(* Logix 5000 project; controller reports 1756-L63 rev 20.11; software revision 20.04; part 3 of 52 *)

        [200].log_data[5].valid := 1, [200].log_data[6].valid := 1, [200].log_data[7].valid := 1, [200].log_data[8].valid := 1, [200].log_data[9].valid := 1, [200].log_data[10].valid := 1, [200].log_data[11].valid := 1, [200].log_data[12].valid := 1, [200].log_data[13].valid := 1, [200].log_data[14].valid := 1, [200].log_data[15].valid := 1, [200].log_data[16].valid := 1, [200].log_data[17].valid := 1, [200].log_data[18].valid := 1, [200].log_data[19].valid := 1, [200].time.Year := 2023, [200].time.Month := 1, [200].time.Day := 18, [200].time.Hour := 2, [200].time.Minute := 29, [200].time.Second := 59, [201].log_data[0].min := 1.0, [201].log_data[0].max := 1.0, [201].log_data[0].total := 900.0, [201].log_data[0].time := 900.0, [201].log_data[0].minminute := 30, [201].log_data[0].maxminute := 30, [201].log_data[0].valid := 1, [201].log_data[1].valid := 1, [201].log_data[2].valid := 1, [201].log_data[3].valid := 1, [201].log_data[4].valid := 1, [201].log_data[5].valid := 1, [201].log_data[6].valid := 1, [201].log_data[7].valid := 1, [201].log_data[8].valid := 1, [201].log_data[9].valid := 1, [201].log_data[10].valid := 1, [201].log_data[11].valid := 1, [201].log_data[12].valid := 1, [201].log_data[13].valid := 1, [201].log_data[14].valid := 1, [201].log_data[15].valid := 1, [201].log_data[16].valid := 1, [201].log_data[17].valid := 1, [201].log_data[18].valid := 1, [201].log_data[19].valid := 1, [201].time.Year := 2023, [201].time.Month := 1, [201].time.Day := 18, [201].time.Hour := 2, [201].time.Minute := 44, [201].time.Second := 59, [202].log_data[0].min := 1.0, [202].log_data[0].max := 1.0, [202].log_data[0].total := 900.0, [202].log_data[0].time := 900.0, [202].log_data[0].minminute := 45, [202].log_data[0].maxminute := 45, [202].log_data[0].valid := 1,
        [202].log_data[1].valid := 1, [202].log_data[2].valid := 1, [202].log_data[3].valid := 1, [202].log_data[4].valid := 1, [202].log_data[5].valid := 1, [202].log_data[6].valid := 1, [202].log_data[7].valid := 1, [202].log_data[8].valid := 1, [202].log_data[9].valid := 1, [202].log_data[10].valid := 1, [202].log_data[11].valid := 1, [202].log_data[12].valid := 1, [202].log_data[13].valid := 1, [202].log_data[14].valid := 1, [202].log_data[15].valid := 1, [202].log_data[16].valid := 1, [202].log_data[17].valid := 1, [202].log_data[18].valid := 1, [202].log_data[19].valid := 1, [202].time.Year := 2023, [202].time.Month := 1, [202].time.Day := 18, [202].time.Hour := 2, [202].time.Minute := 59, [202].time.Second := 59, [203].log_data[0].min := 1.0, [203].log_data[0].max := 1.0, [203].log_data[0].total := 900.0, [203].log_data[0].time := 900.0, [203].log_data[0].valid := 1, [203].log_data[1].valid := 1, [203].log_data[2].valid := 1, [203].log_data[3].valid := 1, [203].log_data[4].valid := 1, [203].log_data[5].valid := 1, [203].log_data[6].valid := 1, [203].log_data[7].valid := 1, [203].log_data[8].valid := 1, [203].log_data[9].valid := 1, [203].log_data[10].valid := 1, [203].log_data[11].valid := 1, [203].log_data[12].valid := 1, [203].log_data[13].valid := 1, [203].log_data[14].valid := 1, [203].log_data[15].valid := 1, [203].log_data[16].valid := 1, [203].log_data[17].valid := 1, [203].log_data[18].valid := 1, [203].log_data[19].valid := 1, [203].time.Year := 2023, [203].time.Month := 1, [203].time.Day := 18, [203].time.Hour := 3, [203].time.Minute := 14, [203].time.Second := 59, [204].log_data[0].min := 1.0, [204].log_data[0].max := 1.0, [204].log_data[0].total := 900.0, [204].log_data[0].time := 900.0, [204].log_data[0].minminute := 15,
        [204].log_data[0].maxminute := 15, [204].log_data[0].valid := 1, [204].log_data[1].valid := 1, [204].log_data[2].valid := 1, [204].log_data[3].valid := 1, [204].log_data[4].valid := 1, [204].log_data[5].valid := 1, [204].log_data[6].valid := 1, [204].log_data[7].valid := 1, [204].log_data[8].valid := 1, [204].log_data[9].valid := 1, [204].log_data[10].valid := 1, [204].log_data[11].valid := 1, [204].log_data[12].valid := 1, [204].log_data[13].valid := 1, [204].log_data[14].valid := 1, [204].log_data[15].valid := 1, [204].log_data[16].valid := 1, [204].log_data[17].valid := 1, [204].log_data[18].valid := 1, [204].log_data[19].valid := 1, [204].time.Year := 2023, [204].time.Month := 1, [204].time.Day := 18, [204].time.Hour := 3, [204].time.Minute := 29, [204].time.Second := 59, [205].log_data[0].min := 1.0, [205].log_data[0].max := 1.0, [205].log_data[0].total := 900.0, [205].log_data[0].time := 900.0, [205].log_data[0].minminute := 30, [205].log_data[0].maxminute := 30, [205].log_data[0].valid := 1, [205].log_data[1].valid := 1, [205].log_data[2].valid := 1, [205].log_data[3].valid := 1, [205].log_data[4].valid := 1, [205].log_data[5].valid := 1, [205].log_data[6].valid := 1, [205].log_data[7].valid := 1, [205].log_data[8].valid := 1, [205].log_data[9].valid := 1, [205].log_data[10].valid := 1, [205].log_data[11].valid := 1, [205].log_data[12].valid := 1, [205].log_data[13].valid := 1, [205].log_data[14].valid := 1, [205].log_data[15].valid := 1, [205].log_data[16].valid := 1, [205].log_data[17].valid := 1, [205].log_data[18].valid := 1, [205].log_data[19].valid := 1, [205].time.Year := 2023, [205].time.Month := 1, [205].time.Day := 18, [205].time.Hour := 3, [205].time.Minute := 44, [205].time.Second := 59, [206].log_data[0].min := 1.0,
        [206].log_data[0].max := 1.0, [206].log_data[0].total := 900.0, [206].log_data[0].time := 900.0, [206].log_data[0].minminute := 45, [206].log_data[0].maxminute := 45, [206].log_data[0].valid := 1, [206].log_data[1].valid := 1, [206].log_data[2].valid := 1, [206].log_data[3].valid := 1, [206].log_data[4].valid := 1, [206].log_data[5].valid := 1, [206].log_data[6].valid := 1, [206].log_data[7].valid := 1, [206].log_data[8].valid := 1, [206].log_data[9].valid := 1, [206].log_data[10].valid := 1, [206].log_data[11].valid := 1, [206].log_data[12].valid := 1, [206].log_data[13].valid := 1, [206].log_data[14].valid := 1, [206].log_data[15].valid := 1, [206].log_data[16].valid := 1, [206].log_data[17].valid := 1, [206].log_data[18].valid := 1, [206].log_data[19].valid := 1, [206].time.Year := 2023, [206].time.Month := 1, [206].time.Day := 18, [206].time.Hour := 3, [206].time.Minute := 59, [206].time.Second := 59, [207].log_data[0].min := 1.0, [207].log_data[0].max := 1.0, [207].log_data[0].total := 900.0, [207].log_data[0].time := 900.0, [207].log_data[0].valid := 1, [207].log_data[1].valid := 1, [207].log_data[2].valid := 1, [207].log_data[3].valid := 1, [207].log_data[4].valid := 1, [207].log_data[5].valid := 1, [207].log_data[6].valid := 1, [207].log_data[7].valid := 1, [207].log_data[8].valid := 1, [207].log_data[9].valid := 1, [207].log_data[10].valid := 1, [207].log_data[11].valid := 1, [207].log_data[12].valid := 1, [207].log_data[13].valid := 1, [207].log_data[14].valid := 1, [207].log_data[15].valid := 1, [207].log_data[16].valid := 1, [207].log_data[17].valid := 1, [207].log_data[18].valid := 1, [207].log_data[19].valid := 1, [207].time.Year := 2023, [207].time.Month := 1, [207].time.Day := 18, [207].time.Hour := 4, [207].time.Minute := 14,
        [207].time.Second := 59, [208].log_data[0].min := 1.0, [208].log_data[0].max := 1.0, [208].log_data[0].total := 900.0, [208].log_data[0].time := 900.0, [208].log_data[0].minminute := 15, [208].log_data[0].maxminute := 15, [208].log_data[0].valid := 1, [208].log_data[1].valid := 1, [208].log_data[2].valid := 1, [208].log_data[3].valid := 1, [208].log_data[4].valid := 1, [208].log_data[5].valid := 1, [208].log_data[6].valid := 1, [208].log_data[7].valid := 1, [208].log_data[8].valid := 1, [208].log_data[9].valid := 1, [208].log_data[10].valid := 1, [208].log_data[11].valid := 1, [208].log_data[12].valid := 1, [208].log_data[13].valid := 1, [208].log_data[14].valid := 1, [208].log_data[15].valid := 1, [208].log_data[16].valid := 1, [208].log_data[17].valid := 1, [208].log_data[18].valid := 1, [208].log_data[19].valid := 1, [208].time.Year := 2023, [208].time.Month := 1, [208].time.Day := 18, [208].time.Hour := 4, [208].time.Minute := 29, [208].time.Second := 59, [209].log_data[0].min := 1.0, [209].log_data[0].max := 1.0, [209].log_data[0].total := 900.0, [209].log_data[0].time := 900.0, [209].log_data[0].minminute := 30, [209].log_data[0].maxminute := 30, [209].log_data[0].valid := 1, [209].log_data[1].valid := 1, [209].log_data[2].valid := 1, [209].log_data[3].valid := 1, [209].log_data[4].valid := 1, [209].log_data[5].valid := 1, [209].log_data[6].valid := 1, [209].log_data[7].valid := 1, [209].log_data[8].valid := 1, [209].log_data[9].valid := 1, [209].log_data[10].valid := 1, [209].log_data[11].valid := 1, [209].log_data[12].valid := 1, [209].log_data[13].valid := 1, [209].log_data[14].valid := 1, [209].log_data[15].valid := 1, [209].log_data[16].valid := 1, [209].log_data[17].valid := 1, [209].log_data[18].valid := 1, [209].log_data[19].valid := 1, [209].time.Year := 2023,
        [209].time.Month := 1, [209].time.Day := 18, [209].time.Hour := 4, [209].time.Minute := 44, [209].time.Second := 59, [210].log_data[0].min := 1.0, [210].log_data[0].max := 1.0, [210].log_data[0].total := 900.0, [210].log_data[0].time := 900.0, [210].log_data[0].minminute := 45, [210].log_data[0].maxminute := 45, [210].log_data[0].valid := 1, [210].log_data[1].valid := 1, [210].log_data[2].valid := 1, [210].log_data[3].valid := 1, [210].log_data[4].valid := 1, [210].log_data[5].valid := 1, [210].log_data[6].valid := 1, [210].log_data[7].valid := 1, [210].log_data[8].valid := 1, [210].log_data[9].valid := 1, [210].log_data[10].valid := 1, [210].log_data[11].valid := 1, [210].log_data[12].valid := 1, [210].log_data[13].valid := 1, [210].log_data[14].valid := 1, [210].log_data[15].valid := 1, [210].log_data[16].valid := 1, [210].log_data[17].valid := 1, [210].log_data[18].valid := 1, [210].log_data[19].valid := 1, [210].time.Year := 2023, [210].time.Month := 1, [210].time.Day := 18, [210].time.Hour := 4, [210].time.Minute := 59, [210].time.Second := 59, [211].log_data[0].min := 1.0, [211].log_data[0].max := 1.0, [211].log_data[0].total := 900.0, [211].log_data[0].time := 900.0, [211].log_data[0].valid := 1, [211].log_data[1].valid := 1, [211].log_data[2].valid := 1, [211].log_data[3].valid := 1, [211].log_data[4].valid := 1, [211].log_data[5].valid := 1, [211].log_data[6].valid := 1, [211].log_data[7].valid := 1, [211].log_data[8].valid := 1, [211].log_data[9].valid := 1, [211].log_data[10].valid := 1, [211].log_data[11].valid := 1, [211].log_data[12].valid := 1, [211].log_data[13].valid := 1, [211].log_data[14].valid := 1, [211].log_data[15].valid := 1, [211].log_data[16].valid := 1, [211].log_data[17].valid := 1, [211].log_data[18].valid := 1,
        [211].log_data[19].valid := 1, [211].time.Year := 2023, [211].time.Month := 1, [211].time.Day := 18, [211].time.Hour := 5, [211].time.Minute := 14, [211].time.Second := 59, [212].log_data[0].min := 1.0, [212].log_data[0].max := 1.0, [212].log_data[0].total := 900.0, [212].log_data[0].time := 900.0, [212].log_data[0].minminute := 15, [212].log_data[0].maxminute := 15, [212].log_data[0].valid := 1, [212].log_data[1].valid := 1, [212].log_data[2].valid := 1, [212].log_data[3].valid := 1, [212].log_data[4].valid := 1, [212].log_data[5].valid := 1, [212].log_data[6].valid := 1, [212].log_data[7].valid := 1, [212].log_data[8].valid := 1, [212].log_data[9].valid := 1, [212].log_data[10].valid := 1, [212].log_data[11].valid := 1, [212].log_data[12].valid := 1, [212].log_data[13].valid := 1, [212].log_data[14].valid := 1, [212].log_data[15].valid := 1, [212].log_data[16].valid := 1, [212].log_data[17].valid := 1, [212].log_data[18].valid := 1, [212].log_data[19].valid := 1, [212].time.Year := 2023, [212].time.Month := 1, [212].time.Day := 18, [212].time.Hour := 5, [212].time.Minute := 29, [212].time.Second := 59, [213].log_data[0].min := 1.0, [213].log_data[0].max := 1.0, [213].log_data[0].total := 900.0, [213].log_data[0].time := 900.0, [213].log_data[0].minminute := 30, [213].log_data[0].maxminute := 30, [213].log_data[0].valid := 1, [213].log_data[1].valid := 1, [213].log_data[2].valid := 1, [213].log_data[3].valid := 1, [213].log_data[4].valid := 1, [213].log_data[5].valid := 1, [213].log_data[6].valid := 1, [213].log_data[7].valid := 1, [213].log_data[8].valid := 1, [213].log_data[9].valid := 1, [213].log_data[10].valid := 1, [213].log_data[11].valid := 1, [213].log_data[12].valid := 1, [213].log_data[13].valid := 1, [213].log_data[14].valid := 1,
        [213].log_data[15].valid := 1, [213].log_data[16].valid := 1, [213].log_data[17].valid := 1, [213].log_data[18].valid := 1, [213].log_data[19].valid := 1, [213].time.Year := 2023, [213].time.Month := 1, [213].time.Day := 18, [213].time.Hour := 5, [213].time.Minute := 44, [213].time.Second := 59, [214].log_data[0].min := 1.0, [214].log_data[0].max := 1.0, [214].log_data[0].total := 900.0, [214].log_data[0].time := 900.0, [214].log_data[0].minminute := 45, [214].log_data[0].maxminute := 45, [214].log_data[0].valid := 1, [214].log_data[1].valid := 1, [214].log_data[2].valid := 1, [214].log_data[3].valid := 1, [214].log_data[4].valid := 1, [214].log_data[5].valid := 1, [214].log_data[6].valid := 1, [214].log_data[7].valid := 1, [214].log_data[8].valid := 1, [214].log_data[9].valid := 1, [214].log_data[10].valid := 1, [214].log_data[11].valid := 1, [214].log_data[12].valid := 1, [214].log_data[13].valid := 1, [214].log_data[14].valid := 1, [214].log_data[15].valid := 1, [214].log_data[16].valid := 1, [214].log_data[17].valid := 1, [214].log_data[18].valid := 1, [214].log_data[19].valid := 1, [214].time.Year := 2023, [214].time.Month := 1, [214].time.Day := 18, [214].time.Hour := 5, [214].time.Minute := 59, [214].time.Second := 59, [215].log_data[0].min := 1.0, [215].log_data[0].max := 1.0, [215].log_data[0].total := 900.0, [215].log_data[0].time := 900.0, [215].log_data[0].valid := 1, [215].log_data[1].valid := 1, [215].log_data[2].valid := 1, [215].log_data[3].valid := 1, [215].log_data[4].valid := 1, [215].log_data[5].valid := 1, [215].log_data[6].valid := 1, [215].log_data[7].valid := 1, [215].log_data[8].valid := 1, [215].log_data[9].valid := 1, [215].log_data[10].valid := 1, [215].log_data[11].valid := 1, [215].log_data[12].valid := 1,
        [215].log_data[13].valid := 1, [215].log_data[14].valid := 1, [215].log_data[15].valid := 1, [215].log_data[16].valid := 1, [215].log_data[17].valid := 1, [215].log_data[18].valid := 1, [215].log_data[19].valid := 1, [215].time.Year := 2023, [215].time.Month := 1, [215].time.Day := 18, [215].time.Hour := 6, [215].time.Minute := 14, [215].time.Second := 59, [216].log_data[0].min := 1.0, [216].log_data[0].max := 1.0, [216].log_data[0].total := 900.0, [216].log_data[0].time := 900.0, [216].log_data[0].minminute := 15, [216].log_data[0].maxminute := 15, [216].log_data[0].valid := 1, [216].log_data[1].valid := 1, [216].log_data[2].valid := 1, [216].log_data[3].valid := 1, [216].log_data[4].valid := 1, [216].log_data[5].valid := 1, [216].log_data[6].valid := 1, [216].log_data[7].valid := 1, [216].log_data[8].valid := 1, [216].log_data[9].valid := 1, [216].log_data[10].valid := 1, [216].log_data[11].valid := 1, [216].log_data[12].valid := 1, [216].log_data[13].valid := 1, [216].log_data[14].valid := 1, [216].log_data[15].valid := 1, [216].log_data[16].valid := 1, [216].log_data[17].valid := 1, [216].log_data[18].valid := 1, [216].log_data[19].valid := 1, [216].time.Year := 2023, [216].time.Month := 1, [216].time.Day := 18, [216].time.Hour := 6, [216].time.Minute := 29, [216].time.Second := 59, [217].log_data[0].min := 1.0, [217].log_data[0].max := 1.0, [217].log_data[0].total := 900.0, [217].log_data[0].time := 900.0, [217].log_data[0].minminute := 30, [217].log_data[0].maxminute := 30, [217].log_data[0].valid := 1, [217].log_data[1].valid := 1, [217].log_data[2].valid := 1, [217].log_data[3].valid := 1, [217].log_data[4].valid := 1, [217].log_data[5].valid := 1, [217].log_data[6].valid := 1, [217].log_data[7].valid := 1, [217].log_data[8].valid := 1,
        [217].log_data[9].valid := 1, [217].log_data[10].valid := 1, [217].log_data[11].valid := 1, [217].log_data[12].valid := 1, [217].log_data[13].valid := 1, [217].log_data[14].valid := 1, [217].log_data[15].valid := 1, [217].log_data[16].valid := 1, [217].log_data[17].valid := 1, [217].log_data[18].valid := 1, [217].log_data[19].valid := 1, [217].time.Year := 2023, [217].time.Month := 1, [217].time.Day := 18, [217].time.Hour := 6, [217].time.Minute := 44, [217].time.Second := 59, [218].log_data[0].min := 1.0, [218].log_data[0].max := 1.0, [218].log_data[0].total := 900.0, [218].log_data[0].time := 900.0, [218].log_data[0].minminute := 45, [218].log_data[0].maxminute := 45, [218].log_data[0].valid := 1, [218].log_data[1].valid := 1, [218].log_data[2].valid := 1, [218].log_data[3].valid := 1, [218].log_data[4].valid := 1, [218].log_data[5].valid := 1, [218].log_data[6].valid := 1, [218].log_data[7].valid := 1, [218].log_data[8].valid := 1, [218].log_data[9].valid := 1, [218].log_data[10].valid := 1, [218].log_data[11].valid := 1, [218].log_data[12].valid := 1, [218].log_data[13].valid := 1, [218].log_data[14].valid := 1, [218].log_data[15].valid := 1, [218].log_data[16].valid := 1, [218].log_data[17].valid := 1, [218].log_data[18].valid := 1, [218].log_data[19].valid := 1, [218].time.Year := 2023, [218].time.Month := 1, [218].time.Day := 18, [218].time.Hour := 6, [218].time.Minute := 59, [218].time.Second := 59, [219].log_data[0].min := 1.0, [219].log_data[0].max := 1.0, [219].log_data[0].total := 900.0, [219].log_data[0].time := 900.0, [219].log_data[0].valid := 1, [219].log_data[1].valid := 1, [219].log_data[2].valid := 1, [219].log_data[3].valid := 1, [219].log_data[4].valid := 1, [219].log_data[5].valid := 1, [219].log_data[6].valid := 1,
        [219].log_data[7].valid := 1, [219].log_data[8].valid := 1, [219].log_data[9].valid := 1, [219].log_data[10].valid := 1, [219].log_data[11].valid := 1, [219].log_data[12].valid := 1, [219].log_data[13].valid := 1, [219].log_data[14].valid := 1, [219].log_data[15].valid := 1, [219].log_data[16].valid := 1, [219].log_data[17].valid := 1, [219].log_data[18].valid := 1, [219].log_data[19].valid := 1, [219].time.Year := 2023, [219].time.Month := 1, [219].time.Day := 18, [219].time.Hour := 7, [219].time.Minute := 14, [219].time.Second := 59, [220].log_data[0].min := 1.0, [220].log_data[0].max := 1.0, [220].log_data[0].total := 900.0, [220].log_data[0].time := 900.0, [220].log_data[0].minminute := 15, [220].log_data[0].maxminute := 15, [220].log_data[0].valid := 1, [220].log_data[1].valid := 1, [220].log_data[2].valid := 1, [220].log_data[3].valid := 1, [220].log_data[4].valid := 1, [220].log_data[5].valid := 1, [220].log_data[6].valid := 1, [220].log_data[7].valid := 1, [220].log_data[8].valid := 1, [220].log_data[9].valid := 1, [220].log_data[10].valid := 1, [220].log_data[11].valid := 1, [220].log_data[12].valid := 1, [220].log_data[13].valid := 1, [220].log_data[14].valid := 1, [220].log_data[15].valid := 1, [220].log_data[16].valid := 1, [220].log_data[17].valid := 1, [220].log_data[18].valid := 1, [220].log_data[19].valid := 1, [220].time.Year := 2023, [220].time.Month := 1, [220].time.Day := 18, [220].time.Hour := 7, [220].time.Minute := 29, [220].time.Second := 59, [221].log_data[0].min := 1.0, [221].log_data[0].max := 1.0, [221].log_data[0].total := 900.0, [221].log_data[0].time := 900.0, [221].log_data[0].minminute := 30, [221].log_data[0].maxminute := 30, [221].log_data[0].valid := 1, [221].log_data[1].valid := 1, [221].log_data[2].valid := 1,
        [221].log_data[3].valid := 1, [221].log_data[4].valid := 1, [221].log_data[5].valid := 1, [221].log_data[6].valid := 1, [221].log_data[7].valid := 1, [221].log_data[8].valid := 1, [221].log_data[9].valid := 1, [221].log_data[10].valid := 1, [221].log_data[11].valid := 1, [221].log_data[12].valid := 1, [221].log_data[13].valid := 1, [221].log_data[14].valid := 1, [221].log_data[15].valid := 1, [221].log_data[16].valid := 1, [221].log_data[17].valid := 1, [221].log_data[18].valid := 1, [221].log_data[19].valid := 1, [221].time.Year := 2023, [221].time.Month := 1, [221].time.Day := 18, [221].time.Hour := 7, [221].time.Minute := 44, [221].time.Second := 59, [222].log_data[0].min := 1.0, [222].log_data[0].max := 1.0, [222].log_data[0].total := 900.0, [222].log_data[0].time := 900.0, [222].log_data[0].minminute := 45, [222].log_data[0].maxminute := 45, [222].log_data[0].valid := 1, [222].log_data[1].valid := 1, [222].log_data[2].valid := 1, [222].log_data[3].valid := 1, [222].log_data[4].valid := 1, [222].log_data[5].valid := 1, [222].log_data[6].valid := 1, [222].log_data[7].valid := 1, [222].log_data[8].valid := 1, [222].log_data[9].valid := 1, [222].log_data[10].valid := 1, [222].log_data[11].valid := 1, [222].log_data[12].valid := 1, [222].log_data[13].valid := 1, [222].log_data[14].valid := 1, [222].log_data[15].valid := 1, [222].log_data[16].valid := 1, [222].log_data[17].valid := 1, [222].log_data[18].valid := 1, [222].log_data[19].valid := 1, [222].time.Year := 2023, [222].time.Month := 1, [222].time.Day := 18, [222].time.Hour := 7, [222].time.Minute := 59, [222].time.Second := 59, [223].log_data[0].min := 1.0, [223].log_data[0].max := 1.0, [223].log_data[0].total := 899.5, [223].log_data[0].time := 899.5, [223].log_data[0].valid := 1,
        [223].log_data[1].valid := 1, [223].log_data[2].valid := 1, [223].log_data[3].valid := 1, [223].log_data[4].valid := 1, [223].log_data[5].valid := 1, [223].log_data[6].valid := 1, [223].log_data[7].valid := 1, [223].log_data[8].valid := 1, [223].log_data[9].valid := 1, [223].log_data[10].valid := 1, [223].log_data[11].valid := 1, [223].log_data[12].valid := 1, [223].log_data[13].valid := 1, [223].log_data[14].valid := 1, [223].log_data[15].valid := 1, [223].log_data[16].valid := 1, [223].log_data[17].valid := 1, [223].log_data[18].valid := 1, [223].log_data[19].valid := 1, [223].time.Year := 2023, [223].time.Month := 1, [223].time.Day := 18, [223].time.Hour := 8, [223].time.Minute := 14, [223].time.Second := 59, [224].log_data[0].min := 1.0, [224].log_data[0].max := 1.0, [224].log_data[0].total := 900.0, [224].log_data[0].time := 900.0, [224].log_data[0].minminute := 15, [224].log_data[0].maxminute := 15, [224].log_data[0].valid := 1, [224].log_data[1].valid := 1, [224].log_data[2].valid := 1, [224].log_data[3].valid := 1, [224].log_data[4].valid := 1, [224].log_data[5].valid := 1, [224].log_data[6].valid := 1, [224].log_data[7].valid := 1, [224].log_data[8].valid := 1, [224].log_data[9].valid := 1, [224].log_data[10].valid := 1, [224].log_data[11].valid := 1, [224].log_data[12].valid := 1, [224].log_data[13].valid := 1, [224].log_data[14].valid := 1, [224].log_data[15].valid := 1, [224].log_data[16].valid := 1, [224].log_data[17].valid := 1, [224].log_data[18].valid := 1, [224].log_data[19].valid := 1, [224].time.Year := 2023, [224].time.Month := 1, [224].time.Day := 18, [224].time.Hour := 8, [224].time.Minute := 29, [224].time.Second := 59, [225].log_data[0].min := 1.0, [225].log_data[0].max := 1.0, [225].log_data[0].total := 900.0,
        [225].log_data[0].time := 900.0, [225].log_data[0].minminute := 30, [225].log_data[0].maxminute := 30, [225].log_data[0].valid := 1, [225].log_data[1].valid := 1, [225].log_data[2].valid := 1, [225].log_data[3].valid := 1, [225].log_data[4].valid := 1, [225].log_data[5].valid := 1, [225].log_data[6].valid := 1, [225].log_data[7].valid := 1, [225].log_data[8].valid := 1, [225].log_data[9].valid := 1, [225].log_data[10].valid := 1, [225].log_data[11].valid := 1, [225].log_data[12].valid := 1, [225].log_data[13].valid := 1, [225].log_data[14].valid := 1, [225].log_data[15].valid := 1, [225].log_data[16].valid := 1, [225].log_data[17].valid := 1, [225].log_data[18].valid := 1, [225].log_data[19].valid := 1, [225].time.Year := 2023, [225].time.Month := 1, [225].time.Day := 18, [225].time.Hour := 8, [225].time.Minute := 44, [225].time.Second := 59, [226].log_data[0].min := 1.0, [226].log_data[0].max := 1.0, [226].log_data[0].total := 900.0, [226].log_data[0].time := 900.0, [226].log_data[0].minminute := 45, [226].log_data[0].maxminute := 45, [226].log_data[0].valid := 1, [226].log_data[1].valid := 1, [226].log_data[2].valid := 1, [226].log_data[3].valid := 1, [226].log_data[4].valid := 1, [226].log_data[5].valid := 1, [226].log_data[6].valid := 1, [226].log_data[7].valid := 1, [226].log_data[8].valid := 1, [226].log_data[9].valid := 1, [226].log_data[10].valid := 1, [226].log_data[11].valid := 1, [226].log_data[12].valid := 1, [226].log_data[13].valid := 1, [226].log_data[14].valid := 1, [226].log_data[15].valid := 1, [226].log_data[16].valid := 1, [226].log_data[17].valid := 1, [226].log_data[18].valid := 1, [226].log_data[19].valid := 1, [226].time.Year := 2023, [226].time.Month := 1, [226].time.Day := 18, [226].time.Hour := 8, [226].time.Minute := 59,
        [226].time.Second := 59, [227].log_data[0].min := 1.0, [227].log_data[0].max := 1.0, [227].log_data[0].total := 900.0, [227].log_data[0].time := 900.0, [227].log_data[0].valid := 1, [227].log_data[1].valid := 1, [227].log_data[2].valid := 1, [227].log_data[3].valid := 1, [227].log_data[4].valid := 1, [227].log_data[5].valid := 1, [227].log_data[6].valid := 1, [227].log_data[7].valid := 1, [227].log_data[8].valid := 1, [227].log_data[9].valid := 1, [227].log_data[10].valid := 1, [227].log_data[11].valid := 1, [227].log_data[12].valid := 1, [227].log_data[13].valid := 1, [227].log_data[14].valid := 1, [227].log_data[15].valid := 1, [227].log_data[16].valid := 1, [227].log_data[17].valid := 1, [227].log_data[18].valid := 1, [227].log_data[19].valid := 1, [227].time.Year := 2023, [227].time.Month := 1, [227].time.Day := 18, [227].time.Hour := 9, [227].time.Minute := 14, [227].time.Second := 59, [228].log_data[0].min := 1.0, [228].log_data[0].max := 1.0, [228].log_data[0].total := 900.0, [228].log_data[0].time := 900.0, [228].log_data[0].minminute := 15, [228].log_data[0].maxminute := 15, [228].log_data[0].valid := 1, [228].log_data[1].valid := 1, [228].log_data[2].valid := 1, [228].log_data[3].valid := 1, [228].log_data[4].valid := 1, [228].log_data[5].valid := 1, [228].log_data[6].valid := 1, [228].log_data[7].valid := 1, [228].log_data[8].valid := 1, [228].log_data[9].valid := 1, [228].log_data[10].valid := 1, [228].log_data[11].valid := 1, [228].log_data[12].valid := 1, [228].log_data[13].valid := 1, [228].log_data[14].valid := 1, [228].log_data[15].valid := 1, [228].log_data[16].valid := 1, [228].log_data[17].valid := 1, [228].log_data[18].valid := 1, [228].log_data[19].valid := 1, [228].time.Year := 2023, [228].time.Month := 1, [228].time.Day := 18,
        [228].time.Hour := 9, [228].time.Minute := 29, [228].time.Second := 59, [229].log_data[0].min := 1.0, [229].log_data[0].max := 1.0, [229].log_data[0].total := 900.0, [229].log_data[0].time := 900.0, [229].log_data[0].minminute := 30, [229].log_data[0].maxminute := 30, [229].log_data[0].valid := 1, [229].log_data[1].valid := 1, [229].log_data[2].valid := 1, [229].log_data[3].valid := 1, [229].log_data[4].valid := 1, [229].log_data[5].valid := 1, [229].log_data[6].valid := 1, [229].log_data[7].valid := 1, [229].log_data[8].valid := 1, [229].log_data[9].valid := 1, [229].log_data[10].valid := 1, [229].log_data[11].valid := 1, [229].log_data[12].valid := 1, [229].log_data[13].valid := 1, [229].log_data[14].valid := 1, [229].log_data[15].valid := 1, [229].log_data[16].valid := 1, [229].log_data[17].valid := 1, [229].log_data[18].valid := 1, [229].log_data[19].valid := 1, [229].time.Year := 2023, [229].time.Month := 1, [229].time.Day := 18, [229].time.Hour := 9, [229].time.Minute := 44, [229].time.Second := 59, [230].log_data[0].min := 1.0, [230].log_data[0].max := 1.0, [230].log_data[0].total := 900.0, [230].log_data[0].time := 900.0, [230].log_data[0].minminute := 45, [230].log_data[0].maxminute := 45, [230].log_data[0].valid := 1, [230].log_data[1].valid := 1, [230].log_data[2].valid := 1, [230].log_data[3].valid := 1, [230].log_data[4].valid := 1, [230].log_data[5].valid := 1, [230].log_data[6].valid := 1, [230].log_data[7].valid := 1, [230].log_data[8].valid := 1, [230].log_data[9].valid := 1, [230].log_data[10].valid := 1, [230].log_data[11].valid := 1, [230].log_data[12].valid := 1, [230].log_data[13].valid := 1, [230].log_data[14].valid := 1, [230].log_data[15].valid := 1, [230].log_data[16].valid := 1, [230].log_data[17].valid := 1, [230].log_data[18].valid := 1,
        [230].log_data[19].valid := 1, [230].time.Year := 2023, [230].time.Month := 1, [230].time.Day := 18, [230].time.Hour := 9, [230].time.Minute := 59, [230].time.Second := 59, [231].log_data[0].min := 1.0, [231].log_data[0].max := 1.0, [231].log_data[0].total := 900.0, [231].log_data[0].time := 900.0, [231].log_data[0].valid := 1, [231].log_data[1].valid := 1, [231].log_data[2].valid := 1, [231].log_data[3].valid := 1, [231].log_data[4].valid := 1, [231].log_data[5].valid := 1, [231].log_data[6].valid := 1, [231].log_data[7].valid := 1, [231].log_data[8].valid := 1, [231].log_data[9].valid := 1, [231].log_data[10].valid := 1, [231].log_data[11].valid := 1, [231].log_data[12].valid := 1, [231].log_data[13].valid := 1, [231].log_data[14].valid := 1, [231].log_data[15].valid := 1, [231].log_data[16].valid := 1, [231].log_data[17].valid := 1, [231].log_data[18].valid := 1, [231].log_data[19].valid := 1, [231].time.Year := 2023, [231].time.Month := 1, [231].time.Day := 18, [231].time.Hour := 10, [231].time.Minute := 14, [231].time.Second := 59, [232].log_data[0].min := 1.0, [232].log_data[0].max := 1.0, [232].log_data[0].total := 900.0, [232].log_data[0].time := 900.0, [232].log_data[0].minminute := 15, [232].log_data[0].maxminute := 15, [232].log_data[0].valid := 1, [232].log_data[1].valid := 1, [232].log_data[2].valid := 1, [232].log_data[3].valid := 1, [232].log_data[4].valid := 1, [232].log_data[5].valid := 1, [232].log_data[6].valid := 1, [232].log_data[7].valid := 1, [232].log_data[8].valid := 1, [232].log_data[9].valid := 1, [232].log_data[10].valid := 1, [232].log_data[11].valid := 1, [232].log_data[12].valid := 1, [232].log_data[13].valid := 1, [232].log_data[14].valid := 1, [232].log_data[15].valid := 1, [232].log_data[16].valid := 1,
        [232].log_data[17].valid := 1, [232].log_data[18].valid := 1, [232].log_data[19].valid := 1, [232].time.Year := 2023, [232].time.Month := 1, [232].time.Day := 18, [232].time.Hour := 10, [232].time.Minute := 29, [232].time.Second := 59, [233].log_data[0].min := 1.0, [233].log_data[0].max := 1.0, [233].log_data[0].total := 900.0, [233].log_data[0].time := 900.0, [233].log_data[0].minminute := 30, [233].log_data[0].maxminute := 30, [233].log_data[0].valid := 1, [233].log_data[1].valid := 1, [233].log_data[2].valid := 1, [233].log_data[3].valid := 1, [233].log_data[4].valid := 1, [233].log_data[5].valid := 1, [233].log_data[6].valid := 1, [233].log_data[7].valid := 1, [233].log_data[8].valid := 1, [233].log_data[9].valid := 1, [233].log_data[10].valid := 1, [233].log_data[11].valid := 1, [233].log_data[12].valid := 1, [233].log_data[13].valid := 1, [233].log_data[14].valid := 1, [233].log_data[15].valid := 1, [233].log_data[16].valid := 1, [233].log_data[17].valid := 1, [233].log_data[18].valid := 1, [233].log_data[19].valid := 1, [233].time.Year := 2023, [233].time.Month := 1, [233].time.Day := 18, [233].time.Hour := 10, [233].time.Minute := 44, [233].time.Second := 59, [234].log_data[0].min := 1.0, [234].log_data[0].max := 1.0, [234].log_data[0].total := 900.0, [234].log_data[0].time := 900.0, [234].log_data[0].minminute := 45, [234].log_data[0].maxminute := 45, [234].log_data[0].valid := 1, [234].log_data[1].valid := 1, [234].log_data[2].valid := 1, [234].log_data[3].valid := 1, [234].log_data[4].valid := 1, [234].log_data[5].valid := 1, [234].log_data[6].valid := 1, [234].log_data[7].valid := 1, [234].log_data[8].valid := 1, [234].log_data[9].valid := 1, [234].log_data[10].valid := 1, [234].log_data[11].valid := 1, [234].log_data[12].valid := 1,
        [234].log_data[13].valid := 1, [234].log_data[14].valid := 1, [234].log_data[15].valid := 1, [234].log_data[16].valid := 1, [234].log_data[17].valid := 1, [234].log_data[18].valid := 1, [234].log_data[19].valid := 1, [234].time.Year := 2023, [234].time.Month := 1, [234].time.Day := 18, [234].time.Hour := 10, [234].time.Minute := 59, [234].time.Second := 59, [235].log_data[0].min := 1.0, [235].log_data[0].max := 1.0, [235].log_data[0].total := 900.0, [235].log_data[0].time := 900.0, [235].log_data[0].valid := 1, [235].log_data[1].valid := 1, [235].log_data[2].valid := 1, [235].log_data[3].valid := 1, [235].log_data[4].valid := 1, [235].log_data[5].valid := 1, [235].log_data[6].valid := 1, [235].log_data[7].valid := 1, [235].log_data[8].valid := 1, [235].log_data[9].valid := 1, [235].log_data[10].valid := 1, [235].log_data[11].valid := 1, [235].log_data[12].valid := 1, [235].log_data[13].valid := 1, [235].log_data[14].valid := 1, [235].log_data[15].valid := 1, [235].log_data[16].valid := 1, [235].log_data[17].valid := 1, [235].log_data[18].valid := 1, [235].log_data[19].valid := 1, [235].time.Year := 2023, [235].time.Month := 1, [235].time.Day := 18, [235].time.Hour := 11, [235].time.Minute := 14, [235].time.Second := 59, [236].log_data[0].min := 1.0, [236].log_data[0].max := 1.0, [236].log_data[0].total := 900.0, [236].log_data[0].time := 900.0, [236].log_data[0].minminute := 15, [236].log_data[0].maxminute := 15, [236].log_data[0].valid := 1, [236].log_data[1].valid := 1, [236].log_data[2].valid := 1, [236].log_data[3].valid := 1, [236].log_data[4].valid := 1, [236].log_data[5].valid := 1, [236].log_data[6].valid := 1, [236].log_data[7].valid := 1, [236].log_data[8].valid := 1, [236].log_data[9].valid := 1, [236].log_data[10].valid := 1,
        [236].log_data[11].valid := 1, [236].log_data[12].valid := 1, [236].log_data[13].valid := 1, [236].log_data[14].valid := 1, [236].log_data[15].valid := 1, [236].log_data[16].valid := 1, [236].log_data[17].valid := 1, [236].log_data[18].valid := 1, [236].log_data[19].valid := 1, [236].time.Year := 2023, [236].time.Month := 1, [236].time.Day := 18, [236].time.Hour := 11, [236].time.Minute := 29, [236].time.Second := 59, [237].log_data[0].min := 1.0, [237].log_data[0].max := 1.0, [237].log_data[0].total := 900.0, [237].log_data[0].time := 900.0, [237].log_data[0].minminute := 30, [237].log_data[0].maxminute := 30, [237].log_data[0].valid := 1, [237].log_data[1].valid := 1, [237].log_data[2].valid := 1, [237].log_data[3].valid := 1, [237].log_data[4].valid := 1, [237].log_data[5].valid := 1, [237].log_data[6].valid := 1, [237].log_data[7].valid := 1, [237].log_data[8].valid := 1, [237].log_data[9].valid := 1, [237].log_data[10].valid := 1, [237].log_data[11].valid := 1, [237].log_data[12].valid := 1, [237].log_data[13].valid := 1, [237].log_data[14].valid := 1, [237].log_data[15].valid := 1, [237].log_data[16].valid := 1, [237].log_data[17].valid := 1, [237].log_data[18].valid := 1, [237].log_data[19].valid := 1, [237].time.Year := 2023, [237].time.Month := 1, [237].time.Day := 18, [237].time.Hour := 11, [237].time.Minute := 44, [237].time.Second := 59, [238].log_data[0].min := 1.0, [238].log_data[0].max := 1.0, [238].log_data[0].total := 900.0, [238].log_data[0].time := 900.0, [238].log_data[0].minminute := 45, [238].log_data[0].maxminute := 45, [238].log_data[0].valid := 1, [238].log_data[1].valid := 1, [238].log_data[2].valid := 1, [238].log_data[3].valid := 1, [238].log_data[4].valid := 1, [238].log_data[5].valid := 1, [238].log_data[6].valid := 1,
        [238].log_data[7].valid := 1, [238].log_data[8].valid := 1, [238].log_data[9].valid := 1, [238].log_data[10].valid := 1, [238].log_data[11].valid := 1, [238].log_data[12].valid := 1, [238].log_data[13].valid := 1, [238].log_data[14].valid := 1, [238].log_data[15].valid := 1, [238].log_data[16].valid := 1, [238].log_data[17].valid := 1, [238].log_data[18].valid := 1, [238].log_data[19].valid := 1, [238].time.Year := 2023, [238].time.Month := 1, [238].time.Day := 18, [238].time.Hour := 11, [238].time.Minute := 59, [238].time.Second := 59, [239].log_data[0].min := 1.0, [239].log_data[0].max := 1.0, [239].log_data[0].total := 900.0, [239].log_data[0].time := 900.0, [239].log_data[0].valid := 1, [239].log_data[1].valid := 1, [239].log_data[2].valid := 1, [239].log_data[3].valid := 1, [239].log_data[4].valid := 1, [239].log_data[5].valid := 1, [239].log_data[6].valid := 1, [239].log_data[7].valid := 1, [239].log_data[8].valid := 1, [239].log_data[9].valid := 1, [239].log_data[10].valid := 1, [239].log_data[11].valid := 1, [239].log_data[12].valid := 1, [239].log_data[13].valid := 1, [239].log_data[14].valid := 1, [239].log_data[15].valid := 1, [239].log_data[16].valid := 1, [239].log_data[17].valid := 1, [239].log_data[18].valid := 1, [239].log_data[19].valid := 1, [239].time.Year := 2023, [239].time.Month := 1, [239].time.Day := 18, [239].time.Hour := 12, [239].time.Minute := 14, [239].time.Second := 59, [240].log_data[0].min := 1.0, [240].log_data[0].max := 1.0, [240].log_data[0].total := 900.0, [240].log_data[0].time := 900.0, [240].log_data[0].minminute := 15, [240].log_data[0].maxminute := 15, [240].log_data[0].valid := 1, [240].log_data[1].valid := 1, [240].log_data[2].valid := 1, [240].log_data[3].valid := 1, [240].log_data[4].valid := 1,
        [240].log_data[5].valid := 1, [240].log_data[6].valid := 1, [240].log_data[7].valid := 1, [240].log_data[8].valid := 1, [240].log_data[9].valid := 1, [240].log_data[10].valid := 1, [240].log_data[11].valid := 1, [240].log_data[12].valid := 1, [240].log_data[13].valid := 1, [240].log_data[14].valid := 1, [240].log_data[15].valid := 1, [240].log_data[16].valid := 1, [240].log_data[17].valid := 1, [240].log_data[18].valid := 1, [240].log_data[19].valid := 1, [240].time.Year := 2023, [240].time.Month := 1, [240].time.Day := 18, [240].time.Hour := 12, [240].time.Minute := 29, [240].time.Second := 59, [241].log_data[0].min := 1.0, [241].log_data[0].max := 1.0, [241].log_data[0].total := 900.0, [241].log_data[0].time := 900.0, [241].log_data[0].minminute := 30, [241].log_data[0].maxminute := 30, [241].log_data[0].valid := 1, [241].log_data[1].valid := 1, [241].log_data[2].valid := 1, [241].log_data[3].valid := 1, [241].log_data[4].valid := 1, [241].log_data[5].valid := 1, [241].log_data[6].valid := 1, [241].log_data[7].valid := 1, [241].log_data[8].valid := 1, [241].log_data[9].valid := 1, [241].log_data[10].valid := 1, [241].log_data[11].valid := 1, [241].log_data[12].valid := 1, [241].log_data[13].valid := 1, [241].log_data[14].valid := 1, [241].log_data[15].valid := 1, [241].log_data[16].valid := 1, [241].log_data[17].valid := 1, [241].log_data[18].valid := 1, [241].log_data[19].valid := 1, [241].time.Year := 2023, [241].time.Month := 1, [241].time.Day := 18, [241].time.Hour := 12, [241].time.Minute := 44, [241].time.Second := 59, [242].log_data[0].min := 1.0, [242].log_data[0].max := 1.0, [242].log_data[0].total := 900.0, [242].log_data[0].time := 900.0, [242].log_data[0].minminute := 45, [242].log_data[0].maxminute := 45, [242].log_data[0].valid := 1,
        [242].log_data[1].valid := 1, [242].log_data[2].valid := 1, [242].log_data[3].valid := 1, [242].log_data[4].valid := 1, [242].log_data[5].valid := 1, [242].log_data[6].valid := 1, [242].log_data[7].valid := 1, [242].log_data[8].valid := 1, [242].log_data[9].valid := 1, [242].log_data[10].valid := 1, [242].log_data[11].valid := 1, [242].log_data[12].valid := 1, [242].log_data[13].valid := 1, [242].log_data[14].valid := 1, [242].log_data[15].valid := 1, [242].log_data[16].valid := 1, [242].log_data[17].valid := 1, [242].log_data[18].valid := 1, [242].log_data[19].valid := 1, [242].time.Year := 2023, [242].time.Month := 1, [242].time.Day := 18, [242].time.Hour := 12, [242].time.Minute := 59, [242].time.Second := 59, [243].log_data[0].min := 1.0, [243].log_data[0].max := 1.0, [243].log_data[0].total := 900.0, [243].log_data[0].time := 900.0, [243].log_data[0].valid := 1, [243].log_data[1].valid := 1, [243].log_data[2].valid := 1, [243].log_data[3].valid := 1, [243].log_data[4].valid := 1, [243].log_data[5].valid := 1, [243].log_data[6].valid := 1, [243].log_data[7].valid := 1, [243].log_data[8].valid := 1, [243].log_data[9].valid := 1, [243].log_data[10].valid := 1, [243].log_data[11].valid := 1, [243].log_data[12].valid := 1, [243].log_data[13].valid := 1, [243].log_data[14].valid := 1, [243].log_data[15].valid := 1, [243].log_data[16].valid := 1, [243].log_data[17].valid := 1, [243].log_data[18].valid := 1, [243].log_data[19].valid := 1, [243].time.Year := 2023, [243].time.Month := 1, [243].time.Day := 18, [243].time.Hour := 13, [243].time.Minute := 14, [243].time.Second := 59, [244].log_data[0].min := 1.0, [244].log_data[0].max := 1.0, [244].log_data[0].total := 900.0, [244].log_data[0].time := 900.0, [244].log_data[0].minminute := 15,
        [244].log_data[0].maxminute := 15, [244].log_data[0].valid := 1, [244].log_data[1].valid := 1, [244].log_data[2].valid := 1, [244].log_data[3].valid := 1, [244].log_data[4].valid := 1, [244].log_data[5].valid := 1, [244].log_data[6].valid := 1, [244].log_data[7].valid := 1, [244].log_data[8].valid := 1, [244].log_data[9].valid := 1, [244].log_data[10].valid := 1, [244].log_data[11].valid := 1, [244].log_data[12].valid := 1, [244].log_data[13].valid := 1, [244].log_data[14].valid := 1, [244].log_data[15].valid := 1, [244].log_data[16].valid := 1, [244].log_data[17].valid := 1, [244].log_data[18].valid := 1, [244].log_data[19].valid := 1, [244].time.Year := 2023, [244].time.Month := 1, [244].time.Day := 18, [244].time.Hour := 13, [244].time.Minute := 29, [244].time.Second := 59, [245].log_data[0].min := 1.0, [245].log_data[0].max := 1.0, [245].log_data[0].total := 900.0, [245].log_data[0].time := 900.0, [245].log_data[0].minminute := 30, [245].log_data[0].maxminute := 30, [245].log_data[0].valid := 1, [245].log_data[1].valid := 1, [245].log_data[2].valid := 1, [245].log_data[3].valid := 1, [245].log_data[4].valid := 1, [245].log_data[5].valid := 1, [245].log_data[6].valid := 1, [245].log_data[7].valid := 1, [245].log_data[8].valid := 1, [245].log_data[9].valid := 1, [245].log_data[10].valid := 1, [245].log_data[11].valid := 1, [245].log_data[12].valid := 1, [245].log_data[13].valid := 1, [245].log_data[14].valid := 1, [245].log_data[15].valid := 1, [245].log_data[16].valid := 1, [245].log_data[17].valid := 1, [245].log_data[18].valid := 1, [245].log_data[19].valid := 1, [245].time.Year := 2023, [245].time.Month := 1, [245].time.Day := 18, [245].time.Hour := 13, [245].time.Minute := 44, [245].time.Second := 59, [246].log_data[0].min := 1.0,
        [246].log_data[0].max := 1.0, [246].log_data[0].total := 900.0, [246].log_data[0].time := 900.0, [246].log_data[0].minminute := 45, [246].log_data[0].maxminute := 45, [246].log_data[0].valid := 1, [246].log_data[1].valid := 1, [246].log_data[2].valid := 1, [246].log_data[3].valid := 1, [246].log_data[4].valid := 1, [246].log_data[5].valid := 1, [246].log_data[6].valid := 1, [246].log_data[7].valid := 1, [246].log_data[8].valid := 1, [246].log_data[9].valid := 1, [246].log_data[10].valid := 1, [246].log_data[11].valid := 1, [246].log_data[12].valid := 1, [246].log_data[13].valid := 1, [246].log_data[14].valid := 1, [246].log_data[15].valid := 1, [246].log_data[16].valid := 1, [246].log_data[17].valid := 1, [246].log_data[18].valid := 1, [246].log_data[19].valid := 1, [246].time.Year := 2023, [246].time.Month := 1, [246].time.Day := 18, [246].time.Hour := 13, [246].time.Minute := 59, [246].time.Second := 59, [247].log_data[0].min := 1.0, [247].log_data[0].max := 1.0, [247].log_data[0].total := 900.0, [247].log_data[0].time := 900.0, [247].log_data[0].valid := 1, [247].log_data[1].valid := 1, [247].log_data[2].valid := 1, [247].log_data[3].valid := 1, [247].log_data[4].valid := 1, [247].log_data[5].valid := 1, [247].log_data[6].valid := 1, [247].log_data[7].valid := 1, [247].log_data[8].valid := 1, [247].log_data[9].valid := 1, [247].log_data[10].valid := 1, [247].log_data[11].valid := 1, [247].log_data[12].valid := 1, [247].log_data[13].valid := 1, [247].log_data[14].valid := 1, [247].log_data[15].valid := 1, [247].log_data[16].valid := 1, [247].log_data[17].valid := 1, [247].log_data[18].valid := 1, [247].log_data[19].valid := 1, [247].time.Year := 2023, [247].time.Month := 1, [247].time.Day := 18, [247].time.Hour := 14, [247].time.Minute := 14,
        [247].time.Second := 59, [248].log_data[0].min := 1.0, [248].log_data[0].max := 1.0, [248].log_data[0].total := 900.0, [248].log_data[0].time := 900.0, [248].log_data[0].minminute := 15, [248].log_data[0].maxminute := 15, [248].log_data[0].valid := 1, [248].log_data[1].valid := 1, [248].log_data[2].valid := 1, [248].log_data[3].valid := 1, [248].log_data[4].valid := 1, [248].log_data[5].valid := 1, [248].log_data[6].valid := 1, [248].log_data[7].valid := 1, [248].log_data[8].valid := 1, [248].log_data[9].valid := 1, [248].log_data[10].valid := 1, [248].log_data[11].valid := 1, [248].log_data[12].valid := 1, [248].log_data[13].valid := 1, [248].log_data[14].valid := 1, [248].log_data[15].valid := 1, [248].log_data[16].valid := 1, [248].log_data[17].valid := 1, [248].log_data[18].valid := 1, [248].log_data[19].valid := 1, [248].time.Year := 2023, [248].time.Month := 1, [248].time.Day := 18, [248].time.Hour := 14, [248].time.Minute := 29, [248].time.Second := 59, [249].log_data[0].min := 1.0, [249].log_data[0].max := 1.0, [249].log_data[0].total := 900.0, [249].log_data[0].time := 900.0, [249].log_data[0].minminute := 30, [249].log_data[0].maxminute := 30, [249].log_data[0].valid := 1, [249].log_data[1].valid := 1, [249].log_data[2].valid := 1, [249].log_data[3].valid := 1, [249].log_data[4].valid := 1, [249].log_data[5].valid := 1, [249].log_data[6].valid := 1, [249].log_data[7].valid := 1, [249].log_data[8].valid := 1, [249].log_data[9].valid := 1, [249].log_data[10].valid := 1, [249].log_data[11].valid := 1, [249].log_data[12].valid := 1, [249].log_data[13].valid := 1, [249].log_data[14].valid := 1, [249].log_data[15].valid := 1, [249].log_data[16].valid := 1, [249].log_data[17].valid := 1, [249].log_data[18].valid := 1, [249].log_data[19].valid := 1, [249].time.Year := 2023,
        [249].time.Month := 1, [249].time.Day := 18, [249].time.Hour := 14, [249].time.Minute := 44, [249].time.Second := 59, [250].log_data[0].min := 1.0, [250].log_data[0].max := 1.0, [250].log_data[0].total := 900.0, [250].log_data[0].time := 900.0, [250].log_data[0].minminute := 45, [250].log_data[0].maxminute := 45, [250].log_data[0].valid := 1, [250].log_data[1].valid := 1, [250].log_data[2].valid := 1, [250].log_data[3].valid := 1, [250].log_data[4].valid := 1, [250].log_data[5].valid := 1, [250].log_data[6].valid := 1, [250].log_data[7].valid := 1, [250].log_data[8].valid := 1, [250].log_data[9].valid := 1, [250].log_data[10].valid := 1, [250].log_data[11].valid := 1, [250].log_data[12].valid := 1, [250].log_data[13].valid := 1, [250].log_data[14].valid := 1, [250].log_data[15].valid := 1, [250].log_data[16].valid := 1, [250].log_data[17].valid := 1, [250].log_data[18].valid := 1, [250].log_data[19].valid := 1, [250].time.Year := 2023, [250].time.Month := 1, [250].time.Day := 18, [250].time.Hour := 14, [250].time.Minute := 59, [250].time.Second := 59, [251].log_data[0].min := 1.0, [251].log_data[0].max := 1.0, [251].log_data[0].total := 900.0, [251].log_data[0].time := 900.0, [251].log_data[0].valid := 1, [251].log_data[1].valid := 1, [251].log_data[2].valid := 1, [251].log_data[3].valid := 1, [251].log_data[4].valid := 1, [251].log_data[5].valid := 1, [251].log_data[6].valid := 1, [251].log_data[7].valid := 1, [251].log_data[8].valid := 1, [251].log_data[9].valid := 1, [251].log_data[10].valid := 1, [251].log_data[11].valid := 1, [251].log_data[12].valid := 1, [251].log_data[13].valid := 1, [251].log_data[14].valid := 1, [251].log_data[15].valid := 1, [251].log_data[16].valid := 1, [251].log_data[17].valid := 1, [251].log_data[18].valid := 1,
        [251].log_data[19].valid := 1, [251].time.Year := 2023, [251].time.Month := 1, [251].time.Day := 18, [251].time.Hour := 15, [251].time.Minute := 14, [251].time.Second := 59, [252].log_data[0].min := 1.0, [252].log_data[0].max := 1.0, [252].log_data[0].total := 900.0, [252].log_data[0].time := 900.0, [252].log_data[0].minminute := 15, [252].log_data[0].maxminute := 15, [252].log_data[0].valid := 1, [252].log_data[1].valid := 1, [252].log_data[2].valid := 1, [252].log_data[3].valid := 1, [252].log_data[4].valid := 1, [252].log_data[5].valid := 1, [252].log_data[6].valid := 1, [252].log_data[7].valid := 1, [252].log_data[8].valid := 1, [252].log_data[9].valid := 1, [252].log_data[10].valid := 1, [252].log_data[11].valid := 1, [252].log_data[12].valid := 1, [252].log_data[13].valid := 1, [252].log_data[14].valid := 1, [252].log_data[15].valid := 1, [252].log_data[16].valid := 1, [252].log_data[17].valid := 1, [252].log_data[18].valid := 1, [252].log_data[19].valid := 1, [252].time.Year := 2023, [252].time.Month := 1, [252].time.Day := 18, [252].time.Hour := 15, [252].time.Minute := 29, [252].time.Second := 59, [253].log_data[0].min := 1.0, [253].log_data[0].max := 1.0, [253].log_data[0].total := 900.0, [253].log_data[0].time := 900.0, [253].log_data[0].minminute := 30, [253].log_data[0].maxminute := 30, [253].log_data[0].valid := 1, [253].log_data[1].valid := 1, [253].log_data[2].valid := 1, [253].log_data[3].valid := 1, [253].log_data[4].valid := 1, [253].log_data[5].valid := 1, [253].log_data[6].valid := 1, [253].log_data[7].valid := 1, [253].log_data[8].valid := 1, [253].log_data[9].valid := 1, [253].log_data[10].valid := 1, [253].log_data[11].valid := 1, [253].log_data[12].valid := 1, [253].log_data[13].valid := 1, [253].log_data[14].valid := 1,
        [253].log_data[15].valid := 1, [253].log_data[16].valid := 1, [253].log_data[17].valid := 1, [253].log_data[18].valid := 1, [253].log_data[19].valid := 1, [253].time.Year := 2023, [253].time.Month := 1, [253].time.Day := 18, [253].time.Hour := 15, [253].time.Minute := 44, [253].time.Second := 59, [254].log_data[0].min := 1.0, [254].log_data[0].max := 1.0, [254].log_data[0].total := 900.0, [254].log_data[0].time := 900.0, [254].log_data[0].minminute := 45, [254].log_data[0].maxminute := 45, [254].log_data[0].valid := 1, [254].log_data[1].valid := 1, [254].log_data[2].valid := 1, [254].log_data[3].valid := 1, [254].log_data[4].valid := 1, [254].log_data[5].valid := 1, [254].log_data[6].valid := 1, [254].log_data[7].valid := 1, [254].log_data[8].valid := 1, [254].log_data[9].valid := 1, [254].log_data[10].valid := 1, [254].log_data[11].valid := 1, [254].log_data[12].valid := 1, [254].log_data[13].valid := 1, [254].log_data[14].valid := 1, [254].log_data[15].valid := 1, [254].log_data[16].valid := 1, [254].log_data[17].valid := 1, [254].log_data[18].valid := 1, [254].log_data[19].valid := 1, [254].time.Year := 2023, [254].time.Month := 1, [254].time.Day := 18, [254].time.Hour := 15, [254].time.Minute := 59, [254].time.Second := 59, [255].log_data[0].min := 1.0, [255].log_data[0].max := 1.0, [255].log_data[0].total := 900.0, [255].log_data[0].time := 900.0, [255].log_data[0].valid := 1, [255].log_data[1].valid := 1, [255].log_data[2].valid := 1, [255].log_data[3].valid := 1, [255].log_data[4].valid := 1, [255].log_data[5].valid := 1, [255].log_data[6].valid := 1, [255].log_data[7].valid := 1, [255].log_data[8].valid := 1, [255].log_data[9].valid := 1, [255].log_data[10].valid := 1, [255].log_data[11].valid := 1, [255].log_data[12].valid := 1,
        [255].log_data[13].valid := 1, [255].log_data[14].valid := 1, [255].log_data[15].valid := 1, [255].log_data[16].valid := 1, [255].log_data[17].valid := 1, [255].log_data[18].valid := 1, [255].log_data[19].valid := 1, [255].time.Year := 2023, [255].time.Month := 1, [255].time.Day := 18, [255].time.Hour := 16, [255].time.Minute := 14, [255].time.Second := 59, [256].log_data[0].min := 1.0, [256].log_data[0].max := 1.0, [256].log_data[0].total := 900.0, [256].log_data[0].time := 900.0, [256].log_data[0].minminute := 15, [256].log_data[0].maxminute := 15, [256].log_data[0].valid := 1, [256].log_data[1].valid := 1, [256].log_data[2].valid := 1, [256].log_data[3].valid := 1, [256].log_data[4].valid := 1, [256].log_data[5].valid := 1, [256].log_data[6].valid := 1, [256].log_data[7].valid := 1, [256].log_data[8].valid := 1, [256].log_data[9].valid := 1, [256].log_data[10].valid := 1, [256].log_data[11].valid := 1, [256].log_data[12].valid := 1, [256].log_data[13].valid := 1, [256].log_data[14].valid := 1, [256].log_data[15].valid := 1, [256].log_data[16].valid := 1, [256].log_data[17].valid := 1, [256].log_data[18].valid := 1, [256].log_data[19].valid := 1, [256].time.Year := 2023, [256].time.Month := 1, [256].time.Day := 18, [256].time.Hour := 16, [256].time.Minute := 29, [256].time.Second := 59, [257].log_data[0].min := 1.0, [257].log_data[0].max := 1.0, [257].log_data[0].total := 900.0, [257].log_data[0].time := 900.0, [257].log_data[0].minminute := 30, [257].log_data[0].maxminute := 30, [257].log_data[0].valid := 1, [257].log_data[1].valid := 1, [257].log_data[2].valid := 1, [257].log_data[3].valid := 1, [257].log_data[4].valid := 1, [257].log_data[5].valid := 1, [257].log_data[6].valid := 1, [257].log_data[7].valid := 1, [257].log_data[8].valid := 1,
        [257].log_data[9].valid := 1, [257].log_data[10].valid := 1, [257].log_data[11].valid := 1, [257].log_data[12].valid := 1, [257].log_data[13].valid := 1, [257].log_data[14].valid := 1, [257].log_data[15].valid := 1, [257].log_data[16].valid := 1, [257].log_data[17].valid := 1, [257].log_data[18].valid := 1, [257].log_data[19].valid := 1, [257].time.Year := 2023, [257].time.Month := 1, [257].time.Day := 18, [257].time.Hour := 16, [257].time.Minute := 44, [257].time.Second := 59, [258].log_data[0].min := 1.0, [258].log_data[0].max := 1.0, [258].log_data[0].total := 900.0, [258].log_data[0].time := 900.0, [258].log_data[0].minminute := 45, [258].log_data[0].maxminute := 45, [258].log_data[0].valid := 1, [258].log_data[1].valid := 1, [258].log_data[2].valid := 1, [258].log_data[3].valid := 1, [258].log_data[4].valid := 1, [258].log_data[5].valid := 1, [258].log_data[6].valid := 1, [258].log_data[7].valid := 1, [258].log_data[8].valid := 1, [258].log_data[9].valid := 1, [258].log_data[10].valid := 1, [258].log_data[11].valid := 1, [258].log_data[12].valid := 1, [258].log_data[13].valid := 1, [258].log_data[14].valid := 1, [258].log_data[15].valid := 1, [258].log_data[16].valid := 1, [258].log_data[17].valid := 1, [258].log_data[18].valid := 1, [258].log_data[19].valid := 1, [258].time.Year := 2023, [258].time.Month := 1, [258].time.Day := 18, [258].time.Hour := 16, [258].time.Minute := 59, [258].time.Second := 59, [259].log_data[0].min := 1.0, [259].log_data[0].max := 1.0, [259].log_data[0].total := 900.0, [259].log_data[0].time := 900.0, [259].log_data[0].valid := 1, [259].log_data[1].valid := 1, [259].log_data[2].valid := 1, [259].log_data[3].valid := 1, [259].log_data[4].valid := 1, [259].log_data[5].valid := 1, [259].log_data[6].valid := 1,
        [259].log_data[7].valid := 1, [259].log_data[8].valid := 1, [259].log_data[9].valid := 1, [259].log_data[10].valid := 1, [259].log_data[11].valid := 1, [259].log_data[12].valid := 1, [259].log_data[13].valid := 1, [259].log_data[14].valid := 1, [259].log_data[15].valid := 1, [259].log_data[16].valid := 1, [259].log_data[17].valid := 1, [259].log_data[18].valid := 1, [259].log_data[19].valid := 1, [259].time.Year := 2023, [259].time.Month := 1, [259].time.Day := 18, [259].time.Hour := 17, [259].time.Minute := 14, [259].time.Second := 59, [260].log_data[0].min := 1.0, [260].log_data[0].max := 1.0, [260].log_data[0].total := 900.0, [260].log_data[0].time := 900.0, [260].log_data[0].minminute := 15, [260].log_data[0].maxminute := 15, [260].log_data[0].valid := 1, [260].log_data[1].valid := 1, [260].log_data[2].valid := 1, [260].log_data[3].valid := 1, [260].log_data[4].valid := 1, [260].log_data[5].valid := 1, [260].log_data[6].valid := 1, [260].log_data[7].valid := 1, [260].log_data[8].valid := 1, [260].log_data[9].valid := 1, [260].log_data[10].valid := 1, [260].log_data[11].valid := 1, [260].log_data[12].valid := 1, [260].log_data[13].valid := 1, [260].log_data[14].valid := 1, [260].log_data[15].valid := 1, [260].log_data[16].valid := 1, [260].log_data[17].valid := 1, [260].log_data[18].valid := 1, [260].log_data[19].valid := 1, [260].time.Year := 2023, [260].time.Month := 1, [260].time.Day := 18, [260].time.Hour := 17, [260].time.Minute := 29, [260].time.Second := 59, [261].log_data[0].min := 1.0, [261].log_data[0].max := 1.0, [261].log_data[0].total := 900.0, [261].log_data[0].time := 900.0, [261].log_data[0].minminute := 30, [261].log_data[0].maxminute := 30, [261].log_data[0].valid := 1, [261].log_data[1].valid := 1, [261].log_data[2].valid := 1,
        [261].log_data[3].valid := 1, [261].log_data[4].valid := 1, [261].log_data[5].valid := 1, [261].log_data[6].valid := 1, [261].log_data[7].valid := 1, [261].log_data[8].valid := 1, [261].log_data[9].valid := 1, [261].log_data[10].valid := 1, [261].log_data[11].valid := 1, [261].log_data[12].valid := 1, [261].log_data[13].valid := 1, [261].log_data[14].valid := 1, [261].log_data[15].valid := 1, [261].log_data[16].valid := 1, [261].log_data[17].valid := 1, [261].log_data[18].valid := 1, [261].log_data[19].valid := 1, [261].time.Year := 2023, [261].time.Month := 1, [261].time.Day := 18, [261].time.Hour := 17, [261].time.Minute := 44, [261].time.Second := 59, [262].log_data[0].min := 1.0, [262].log_data[0].max := 1.0, [262].log_data[0].total := 900.0, [262].log_data[0].time := 900.0, [262].log_data[0].minminute := 45, [262].log_data[0].maxminute := 45, [262].log_data[0].valid := 1, [262].log_data[1].valid := 1, [262].log_data[2].valid := 1, [262].log_data[3].valid := 1, [262].log_data[4].valid := 1, [262].log_data[5].valid := 1, [262].log_data[6].valid := 1, [262].log_data[7].valid := 1, [262].log_data[8].valid := 1, [262].log_data[9].valid := 1, [262].log_data[10].valid := 1, [262].log_data[11].valid := 1, [262].log_data[12].valid := 1, [262].log_data[13].valid := 1, [262].log_data[14].valid := 1, [262].log_data[15].valid := 1, [262].log_data[16].valid := 1, [262].log_data[17].valid := 1, [262].log_data[18].valid := 1, [262].log_data[19].valid := 1, [262].time.Year := 2023, [262].time.Month := 1, [262].time.Day := 18, [262].time.Hour := 17, [262].time.Minute := 59, [262].time.Second := 59, [263].log_data[0].min := 1.0, [263].log_data[0].max := 1.0, [263].log_data[0].total := 900.0, [263].log_data[0].time := 900.0, [263].log_data[0].valid := 1,
        [263].log_data[1].valid := 1, [263].log_data[2].valid := 1, [263].log_data[3].valid := 1, [263].log_data[4].valid := 1, [263].log_data[5].valid := 1, [263].log_data[6].valid := 1, [263].log_data[7].valid := 1, [263].log_data[8].valid := 1, [263].log_data[9].valid := 1, [263].log_data[10].valid := 1, [263].log_data[11].valid := 1, [263].log_data[12].valid := 1, [263].log_data[13].valid := 1, [263].log_data[14].valid := 1, [263].log_data[15].valid := 1, [263].log_data[16].valid := 1, [263].log_data[17].valid := 1, [263].log_data[18].valid := 1, [263].log_data[19].valid := 1, [263].time.Year := 2023, [263].time.Month := 1, [263].time.Day := 18, [263].time.Hour := 18, [263].time.Minute := 14, [263].time.Second := 59, [264].log_data[0].min := 1.0, [264].log_data[0].max := 1.0, [264].log_data[0].total := 900.0, [264].log_data[0].time := 900.0, [264].log_data[0].minminute := 15, [264].log_data[0].maxminute := 15, [264].log_data[0].valid := 1, [264].log_data[1].valid := 1, [264].log_data[2].valid := 1, [264].log_data[3].valid := 1, [264].log_data[4].valid := 1, [264].log_data[5].valid := 1, [264].log_data[6].valid := 1, [264].log_data[7].valid := 1, [264].log_data[8].valid := 1, [264].log_data[9].valid := 1, [264].log_data[10].valid := 1, [264].log_data[11].valid := 1, [264].log_data[12].valid := 1, [264].log_data[13].valid := 1, [264].log_data[14].valid := 1, [264].log_data[15].valid := 1, [264].log_data[16].valid := 1, [264].log_data[17].valid := 1, [264].log_data[18].valid := 1, [264].log_data[19].valid := 1, [264].time.Year := 2023, [264].time.Month := 1, [264].time.Day := 18, [264].time.Hour := 18, [264].time.Minute := 29, [264].time.Second := 59, [265].log_data[0].min := 1.0, [265].log_data[0].max := 1.0, [265].log_data[0].total := 900.0,
        [265].log_data[0].time := 900.0, [265].log_data[0].minminute := 30, [265].log_data[0].maxminute := 30, [265].log_data[0].valid := 1, [265].log_data[1].valid := 1, [265].log_data[2].valid := 1, [265].log_data[3].valid := 1, [265].log_data[4].valid := 1, [265].log_data[5].valid := 1, [265].log_data[6].valid := 1, [265].log_data[7].valid := 1, [265].log_data[8].valid := 1, [265].log_data[9].valid := 1, [265].log_data[10].valid := 1, [265].log_data[11].valid := 1, [265].log_data[12].valid := 1, [265].log_data[13].valid := 1, [265].log_data[14].valid := 1, [265].log_data[15].valid := 1, [265].log_data[16].valid := 1, [265].log_data[17].valid := 1, [265].log_data[18].valid := 1, [265].log_data[19].valid := 1, [265].time.Year := 2023, [265].time.Month := 1, [265].time.Day := 18, [265].time.Hour := 18, [265].time.Minute := 44, [265].time.Second := 59, [266].log_data[0].min := 1.0, [266].log_data[0].max := 1.0, [266].log_data[0].total := 900.0, [266].log_data[0].time := 900.0, [266].log_data[0].minminute := 45, [266].log_data[0].maxminute := 45, [266].log_data[0].valid := 1, [266].log_data[1].valid := 1, [266].log_data[2].valid := 1, [266].log_data[3].valid := 1, [266].log_data[4].valid := 1, [266].log_data[5].valid := 1, [266].log_data[6].valid := 1, [266].log_data[7].valid := 1, [266].log_data[8].valid := 1, [266].log_data[9].valid := 1, [266].log_data[10].valid := 1, [266].log_data[11].valid := 1, [266].log_data[12].valid := 1, [266].log_data[13].valid := 1, [266].log_data[14].valid := 1, [266].log_data[15].valid := 1, [266].log_data[16].valid := 1, [266].log_data[17].valid := 1, [266].log_data[18].valid := 1, [266].log_data[19].valid := 1, [266].time.Year := 2023, [266].time.Month := 1, [266].time.Day := 18, [266].time.Hour := 18, [266].time.Minute := 59,
        [266].time.Second := 59, [267].log_data[0].min := 1.0, [267].log_data[0].max := 1.0, [267].log_data[0].total := 900.0, [267].log_data[0].time := 900.0, [267].log_data[0].valid := 1, [267].log_data[1].valid := 1, [267].log_data[2].valid := 1, [267].log_data[3].valid := 1, [267].log_data[4].valid := 1, [267].log_data[5].valid := 1, [267].log_data[6].valid := 1, [267].log_data[7].valid := 1, [267].log_data[8].valid := 1, [267].log_data[9].valid := 1, [267].log_data[10].valid := 1, [267].log_data[11].valid := 1, [267].log_data[12].valid := 1, [267].log_data[13].valid := 1, [267].log_data[14].valid := 1, [267].log_data[15].valid := 1, [267].log_data[16].valid := 1, [267].log_data[17].valid := 1, [267].log_data[18].valid := 1, [267].log_data[19].valid := 1, [267].time.Year := 2023, [267].time.Month := 1, [267].time.Day := 18, [267].time.Hour := 19, [267].time.Minute := 14, [267].time.Second := 59, [268].log_data[0].min := 1.0, [268].log_data[0].max := 1.0, [268].log_data[0].total := 900.0, [268].log_data[0].time := 900.0, [268].log_data[0].minminute := 15, [268].log_data[0].maxminute := 15, [268].log_data[0].valid := 1, [268].log_data[1].valid := 1, [268].log_data[2].valid := 1, [268].log_data[3].valid := 1, [268].log_data[4].valid := 1, [268].log_data[5].valid := 1, [268].log_data[6].valid := 1, [268].log_data[7].valid := 1, [268].log_data[8].valid := 1, [268].log_data[9].valid := 1, [268].log_data[10].valid := 1, [268].log_data[11].valid := 1, [268].log_data[12].valid := 1, [268].log_data[13].valid := 1, [268].log_data[14].valid := 1, [268].log_data[15].valid := 1, [268].log_data[16].valid := 1, [268].log_data[17].valid := 1, [268].log_data[18].valid := 1, [268].log_data[19].valid := 1, [268].time.Year := 2023, [268].time.Month := 1, [268].time.Day := 18,
        [268].time.Hour := 19, [268].time.Minute := 29, [268].time.Second := 59, [269].log_data[0].min := 1.0, [269].log_data[0].max := 1.0, [269].log_data[0].total := 900.0, [269].log_data[0].time := 900.0, [269].log_data[0].minminute := 30, [269].log_data[0].maxminute := 30, [269].log_data[0].valid := 1, [269].log_data[1].valid := 1, [269].log_data[2].valid := 1, [269].log_data[3].valid := 1, [269].log_data[4].valid := 1, [269].log_data[5].valid := 1, [269].log_data[6].valid := 1, [269].log_data[7].valid := 1, [269].log_data[8].valid := 1, [269].log_data[9].valid := 1, [269].log_data[10].valid := 1, [269].log_data[11].valid := 1, [269].log_data[12].valid := 1, [269].log_data[13].valid := 1, [269].log_data[14].valid := 1, [269].log_data[15].valid := 1, [269].log_data[16].valid := 1, [269].log_data[17].valid := 1, [269].log_data[18].valid := 1, [269].log_data[19].valid := 1, [269].time.Year := 2023, [269].time.Month := 1, [269].time.Day := 18, [269].time.Hour := 19, [269].time.Minute := 44, [269].time.Second := 59, [270].log_data[0].min := 1.0, [270].log_data[0].max := 1.0, [270].log_data[0].total := 900.0, [270].log_data[0].time := 900.0, [270].log_data[0].minminute := 45, [270].log_data[0].maxminute := 45, [270].log_data[0].valid := 1, [270].log_data[1].valid := 1, [270].log_data[2].valid := 1, [270].log_data[3].valid := 1, [270].log_data[4].valid := 1, [270].log_data[5].valid := 1, [270].log_data[6].valid := 1, [270].log_data[7].valid := 1, [270].log_data[8].valid := 1, [270].log_data[9].valid := 1, [270].log_data[10].valid := 1, [270].log_data[11].valid := 1, [270].log_data[12].valid := 1, [270].log_data[13].valid := 1, [270].log_data[14].valid := 1, [270].log_data[15].valid := 1, [270].log_data[16].valid := 1, [270].log_data[17].valid := 1, [270].log_data[18].valid := 1,
        [270].log_data[19].valid := 1, [270].time.Year := 2023, [270].time.Month := 1, [270].time.Day := 18, [270].time.Hour := 19, [270].time.Minute := 59, [270].time.Second := 59, [271].log_data[0].min := 1.0, [271].log_data[0].max := 1.0, [271].log_data[0].total := 900.0, [271].log_data[0].time := 900.0, [271].log_data[0].valid := 1, [271].log_data[1].valid := 1, [271].log_data[2].valid := 1, [271].log_data[3].valid := 1, [271].log_data[4].valid := 1, [271].log_data[5].valid := 1, [271].log_data[6].valid := 1, [271].log_data[7].valid := 1, [271].log_data[8].valid := 1, [271].log_data[9].valid := 1, [271].log_data[10].valid := 1, [271].log_data[11].valid := 1, [271].log_data[12].valid := 1, [271].log_data[13].valid := 1, [271].log_data[14].valid := 1, [271].log_data[15].valid := 1, [271].log_data[16].valid := 1, [271].log_data[17].valid := 1, [271].log_data[18].valid := 1, [271].log_data[19].valid := 1, [271].time.Year := 2023, [271].time.Month := 1, [271].time.Day := 18, [271].time.Hour := 20, [271].time.Minute := 14, [271].time.Second := 59, [272].log_data[0].min := 1.0, [272].log_data[0].max := 1.0, [272].log_data[0].total := 900.0, [272].log_data[0].time := 900.0, [272].log_data[0].minminute := 15, [272].log_data[0].maxminute := 15, [272].log_data[0].valid := 1, [272].log_data[1].valid := 1, [272].log_data[2].valid := 1, [272].log_data[3].valid := 1, [272].log_data[4].valid := 1, [272].log_data[5].valid := 1, [272].log_data[6].valid := 1, [272].log_data[7].valid := 1, [272].log_data[8].valid := 1, [272].log_data[9].valid := 1, [272].log_data[10].valid := 1, [272].log_data[11].valid := 1, [272].log_data[12].valid := 1, [272].log_data[13].valid := 1, [272].log_data[14].valid := 1, [272].log_data[15].valid := 1, [272].log_data[16].valid := 1,
        [272].log_data[17].valid := 1, [272].log_data[18].valid := 1, [272].log_data[19].valid := 1, [272].time.Year := 2023, [272].time.Month := 1, [272].time.Day := 18, [272].time.Hour := 20, [272].time.Minute := 29, [272].time.Second := 59, [273].log_data[0].min := 1.0, [273].log_data[0].max := 1.0, [273].log_data[0].total := 900.0, [273].log_data[0].time := 900.0, [273].log_data[0].minminute := 30, [273].log_data[0].maxminute := 30, [273].log_data[0].valid := 1, [273].log_data[1].valid := 1, [273].log_data[2].valid := 1, [273].log_data[3].valid := 1, [273].log_data[4].valid := 1, [273].log_data[5].valid := 1, [273].log_data[6].valid := 1, [273].log_data[7].valid := 1, [273].log_data[8].valid := 1, [273].log_data[9].valid := 1, [273].log_data[10].valid := 1, [273].log_data[11].valid := 1, [273].log_data[12].valid := 1, [273].log_data[13].valid := 1, [273].log_data[14].valid := 1, [273].log_data[15].valid := 1, [273].log_data[16].valid := 1, [273].log_data[17].valid := 1, [273].log_data[18].valid := 1, [273].log_data[19].valid := 1, [273].time.Year := 2023, [273].time.Month := 1, [273].time.Day := 18, [273].time.Hour := 20, [273].time.Minute := 44, [273].time.Second := 59, [274].log_data[0].min := 1.0, [274].log_data[0].max := 1.0, [274].log_data[0].total := 900.0, [274].log_data[0].time := 900.0, [274].log_data[0].minminute := 45, [274].log_data[0].maxminute := 45, [274].log_data[0].valid := 1, [274].log_data[1].valid := 1, [274].log_data[2].valid := 1, [274].log_data[3].valid := 1, [274].log_data[4].valid := 1, [274].log_data[5].valid := 1, [274].log_data[6].valid := 1, [274].log_data[7].valid := 1, [274].log_data[8].valid := 1, [274].log_data[9].valid := 1, [274].log_data[10].valid := 1, [274].log_data[11].valid := 1, [274].log_data[12].valid := 1,
        [274].log_data[13].valid := 1, [274].log_data[14].valid := 1, [274].log_data[15].valid := 1, [274].log_data[16].valid := 1, [274].log_data[17].valid := 1, [274].log_data[18].valid := 1, [274].log_data[19].valid := 1, [274].time.Year := 2023, [274].time.Month := 1, [274].time.Day := 18, [274].time.Hour := 20, [274].time.Minute := 59, [274].time.Second := 59, [275].log_data[0].min := 1.0, [275].log_data[0].max := 1.0, [275].log_data[0].total := 899.5, [275].log_data[0].time := 899.5, [275].log_data[0].valid := 1, [275].log_data[1].valid := 1, [275].log_data[2].valid := 1, [275].log_data[3].valid := 1, [275].log_data[4].valid := 1, [275].log_data[5].valid := 1, [275].log_data[6].valid := 1, [275].log_data[7].valid := 1, [275].log_data[8].valid := 1, [275].log_data[9].valid := 1, [275].log_data[10].valid := 1, [275].log_data[11].valid := 1, [275].log_data[12].valid := 1, [275].log_data[13].valid := 1, [275].log_data[14].valid := 1, [275].log_data[15].valid := 1, [275].log_data[16].valid := 1, [275].log_data[17].valid := 1, [275].log_data[18].valid := 1, [275].log_data[19].valid := 1, [275].time.Year := 2023, [275].time.Month := 1, [275].time.Day := 18, [275].time.Hour := 21, [275].time.Minute := 14, [275].time.Second := 59, [276].log_data[0].min := 1.0, [276].log_data[0].max := 1.0, [276].log_data[0].total := 900.0, [276].log_data[0].time := 900.0, [276].log_data[0].minminute := 15, [276].log_data[0].maxminute := 15, [276].log_data[0].valid := 1, [276].log_data[1].valid := 1, [276].log_data[2].valid := 1, [276].log_data[3].valid := 1, [276].log_data[4].valid := 1, [276].log_data[5].valid := 1, [276].log_data[6].valid := 1, [276].log_data[7].valid := 1, [276].log_data[8].valid := 1, [276].log_data[9].valid := 1, [276].log_data[10].valid := 1,
        [276].log_data[11].valid := 1, [276].log_data[12].valid := 1, [276].log_data[13].valid := 1, [276].log_data[14].valid := 1, [276].log_data[15].valid := 1, [276].log_data[16].valid := 1, [276].log_data[17].valid := 1, [276].log_data[18].valid := 1, [276].log_data[19].valid := 1, [276].time.Year := 2023, [276].time.Month := 1, [276].time.Day := 18, [276].time.Hour := 21, [276].time.Minute := 29, [276].time.Second := 59, [277].log_data[0].min := 1.0, [277].log_data[0].max := 1.0, [277].log_data[0].total := 900.0, [277].log_data[0].time := 900.0, [277].log_data[0].minminute := 30, [277].log_data[0].maxminute := 30, [277].log_data[0].valid := 1, [277].log_data[1].valid := 1, [277].log_data[2].valid := 1, [277].log_data[3].valid := 1, [277].log_data[4].valid := 1, [277].log_data[5].valid := 1, [277].log_data[6].valid := 1, [277].log_data[7].valid := 1, [277].log_data[8].valid := 1, [277].log_data[9].valid := 1, [277].log_data[10].valid := 1, [277].log_data[11].valid := 1, [277].log_data[12].valid := 1, [277].log_data[13].valid := 1, [277].log_data[14].valid := 1, [277].log_data[15].valid := 1, [277].log_data[16].valid := 1, [277].log_data[17].valid := 1, [277].log_data[18].valid := 1, [277].log_data[19].valid := 1, [277].time.Year := 2023, [277].time.Month := 1, [277].time.Day := 18, [277].time.Hour := 21, [277].time.Minute := 44, [277].time.Second := 59, [278].log_data[0].min := 1.0, [278].log_data[0].max := 1.0, [278].log_data[0].total := 900.0, [278].log_data[0].time := 900.0, [278].log_data[0].minminute := 45, [278].log_data[0].maxminute := 45, [278].log_data[0].valid := 1, [278].log_data[1].valid := 1, [278].log_data[2].valid := 1, [278].log_data[3].valid := 1, [278].log_data[4].valid := 1, [278].log_data[5].valid := 1, [278].log_data[6].valid := 1,
        [278].log_data[7].valid := 1, [278].log_data[8].valid := 1, [278].log_data[9].valid := 1, [278].log_data[10].valid := 1, [278].log_data[11].valid := 1, [278].log_data[12].valid := 1, [278].log_data[13].valid := 1, [278].log_data[14].valid := 1, [278].log_data[15].valid := 1, [278].log_data[16].valid := 1, [278].log_data[17].valid := 1, [278].log_data[18].valid := 1, [278].log_data[19].valid := 1, [278].time.Year := 2023, [278].time.Month := 1, [278].time.Day := 18, [278].time.Hour := 21, [278].time.Minute := 59, [278].time.Second := 59, [279].log_data[0].min := 1.0, [279].log_data[0].max := 1.0, [279].log_data[0].total := 900.0, [279].log_data[0].time := 900.0, [279].log_data[0].valid := 1, [279].log_data[1].valid := 1, [279].log_data[2].valid := 1, [279].log_data[3].valid := 1, [279].log_data[4].valid := 1, [279].log_data[5].valid := 1, [279].log_data[6].valid := 1, [279].log_data[7].valid := 1, [279].log_data[8].valid := 1, [279].log_data[9].valid := 1, [279].log_data[10].valid := 1, [279].log_data[11].valid := 1, [279].log_data[12].valid := 1, [279].log_data[13].valid := 1, [279].log_data[14].valid := 1, [279].log_data[15].valid := 1, [279].log_data[16].valid := 1, [279].log_data[17].valid := 1, [279].log_data[18].valid := 1, [279].log_data[19].valid := 1, [279].time.Year := 2023, [279].time.Month := 1, [279].time.Day := 18, [279].time.Hour := 22, [279].time.Minute := 14, [279].time.Second := 59, [280].log_data[0].min := 1.0, [280].log_data[0].max := 1.0, [280].log_data[0].total := 900.0, [280].log_data[0].time := 900.0, [280].log_data[0].minminute := 15, [280].log_data[0].maxminute := 15, [280].log_data[0].valid := 1, [280].log_data[1].valid := 1, [280].log_data[2].valid := 1, [280].log_data[3].valid := 1, [280].log_data[4].valid := 1,
        [280].log_data[5].valid := 1, [280].log_data[6].valid := 1, [280].log_data[7].valid := 1, [280].log_data[8].valid := 1, [280].log_data[9].valid := 1, [280].log_data[10].valid := 1, [280].log_data[11].valid := 1, [280].log_data[12].valid := 1, [280].log_data[13].valid := 1, [280].log_data[14].valid := 1, [280].log_data[15].valid := 1, [280].log_data[16].valid := 1, [280].log_data[17].valid := 1, [280].log_data[18].valid := 1, [280].log_data[19].valid := 1, [280].time.Year := 2023, [280].time.Month := 1, [280].time.Day := 18, [280].time.Hour := 22, [280].time.Minute := 29, [280].time.Second := 59, [281].log_data[0].min := 1.0, [281].log_data[0].max := 1.0, [281].log_data[0].total := 900.0, [281].log_data[0].time := 900.0, [281].log_data[0].minminute := 30, [281].log_data[0].maxminute := 30, [281].log_data[0].valid := 1, [281].log_data[1].valid := 1, [281].log_data[2].valid := 1, [281].log_data[3].valid := 1, [281].log_data[4].valid := 1, [281].log_data[5].valid := 1, [281].log_data[6].valid := 1, [281].log_data[7].valid := 1, [281].log_data[8].valid := 1, [281].log_data[9].valid := 1, [281].log_data[10].valid := 1, [281].log_data[11].valid := 1, [281].log_data[12].valid := 1, [281].log_data[13].valid := 1, [281].log_data[14].valid := 1, [281].log_data[15].valid := 1, [281].log_data[16].valid := 1, [281].log_data[17].valid := 1, [281].log_data[18].valid := 1, [281].log_data[19].valid := 1, [281].time.Year := 2023, [281].time.Month := 1, [281].time.Day := 18, [281].time.Hour := 22, [281].time.Minute := 44, [281].time.Second := 59, [282].log_data[0].min := 1.0, [282].log_data[0].max := 1.0, [282].log_data[0].total := 900.0, [282].log_data[0].time := 900.0, [282].log_data[0].minminute := 45, [282].log_data[0].maxminute := 45, [282].log_data[0].valid := 1,
        [282].log_data[1].valid := 1, [282].log_data[2].valid := 1, [282].log_data[3].valid := 1, [282].log_data[4].valid := 1, [282].log_data[5].valid := 1, [282].log_data[6].valid := 1, [282].log_data[7].valid := 1, [282].log_data[8].valid := 1, [282].log_data[9].valid := 1, [282].log_data[10].valid := 1, [282].log_data[11].valid := 1, [282].log_data[12].valid := 1, [282].log_data[13].valid := 1, [282].log_data[14].valid := 1, [282].log_data[15].valid := 1, [282].log_data[16].valid := 1, [282].log_data[17].valid := 1, [282].log_data[18].valid := 1, [282].log_data[19].valid := 1, [282].time.Year := 2023, [282].time.Month := 1, [282].time.Day := 18, [282].time.Hour := 22, [282].time.Minute := 59, [282].time.Second := 59, [283].log_data[0].min := 1.0, [283].log_data[0].max := 1.0, [283].log_data[0].total := 900.0, [283].log_data[0].time := 900.0, [283].log_data[0].valid := 1, [283].log_data[1].valid := 1, [283].log_data[2].valid := 1, [283].log_data[3].valid := 1, [283].log_data[4].valid := 1, [283].log_data[5].valid := 1, [283].log_data[6].valid := 1, [283].log_data[7].valid := 1, [283].log_data[8].valid := 1, [283].log_data[9].valid := 1, [283].log_data[10].valid := 1, [283].log_data[11].valid := 1, [283].log_data[12].valid := 1, [283].log_data[13].valid := 1, [283].log_data[14].valid := 1, [283].log_data[15].valid := 1, [283].log_data[16].valid := 1, [283].log_data[17].valid := 1, [283].log_data[18].valid := 1, [283].log_data[19].valid := 1, [283].time.Year := 2023, [283].time.Month := 1, [283].time.Day := 18, [283].time.Hour := 23, [283].time.Minute := 14, [283].time.Second := 59, [284].log_data[0].min := 1.0, [284].log_data[0].max := 1.0, [284].log_data[0].total := 900.0, [284].log_data[0].time := 900.0, [284].log_data[0].minminute := 15,
        [284].log_data[0].maxminute := 15, [284].log_data[0].valid := 1, [284].log_data[1].valid := 1, [284].log_data[2].valid := 1, [284].log_data[3].valid := 1, [284].log_data[4].valid := 1, [284].log_data[5].valid := 1, [284].log_data[6].valid := 1, [284].log_data[7].valid := 1, [284].log_data[8].valid := 1, [284].log_data[9].valid := 1, [284].log_data[10].valid := 1, [284].log_data[11].valid := 1, [284].log_data[12].valid := 1, [284].log_data[13].valid := 1, [284].log_data[14].valid := 1, [284].log_data[15].valid := 1, [284].log_data[16].valid := 1, [284].log_data[17].valid := 1, [284].log_data[18].valid := 1, [284].log_data[19].valid := 1, [284].time.Year := 2023, [284].time.Month := 1, [284].time.Day := 18, [284].time.Hour := 23, [284].time.Minute := 29, [284].time.Second := 59, [285].log_data[0].min := 1.0, [285].log_data[0].max := 1.0, [285].log_data[0].total := 900.0, [285].log_data[0].time := 900.0, [285].log_data[0].minminute := 30, [285].log_data[0].maxminute := 30, [285].log_data[0].valid := 1, [285].log_data[1].valid := 1, [285].log_data[2].valid := 1, [285].log_data[3].valid := 1, [285].log_data[4].valid := 1, [285].log_data[5].valid := 1, [285].log_data[6].valid := 1, [285].log_data[7].valid := 1, [285].log_data[8].valid := 1, [285].log_data[9].valid := 1, [285].log_data[10].valid := 1, [285].log_data[11].valid := 1, [285].log_data[12].valid := 1, [285].log_data[13].valid := 1, [285].log_data[14].valid := 1, [285].log_data[15].valid := 1, [285].log_data[16].valid := 1, [285].log_data[17].valid := 1, [285].log_data[18].valid := 1, [285].log_data[19].valid := 1, [285].time.Year := 2023, [285].time.Month := 1, [285].time.Day := 18, [285].time.Hour := 23, [285].time.Minute := 44, [285].time.Second := 59, [286].log_data[0].min := 1.0,
        [286].log_data[0].max := 1.0, [286].log_data[0].total := 900.0, [286].log_data[0].time := 900.0, [286].log_data[0].minminute := 45, [286].log_data[0].maxminute := 45, [286].log_data[0].valid := 1, [286].log_data[1].valid := 1, [286].log_data[2].valid := 1, [286].log_data[3].valid := 1, [286].log_data[4].valid := 1, [286].log_data[5].valid := 1, [286].log_data[6].valid := 1, [286].log_data[7].valid := 1, [286].log_data[8].valid := 1, [286].log_data[9].valid := 1, [286].log_data[10].valid := 1, [286].log_data[11].valid := 1, [286].log_data[12].valid := 1, [286].log_data[13].valid := 1, [286].log_data[14].valid := 1, [286].log_data[15].valid := 1, [286].log_data[16].valid := 1, [286].log_data[17].valid := 1, [286].log_data[18].valid := 1, [286].log_data[19].valid := 1, [286].time.Year := 2023, [286].time.Month := 1, [286].time.Day := 18, [286].time.Hour := 23, [286].time.Minute := 59, [286].time.Second := 59, [287].log_data[0].min := 1.0, [287].log_data[0].max := 1.0, [287].log_data[0].total := 900.0, [287].log_data[0].time := 900.0, [287].log_data[0].valid := 1, [287].log_data[1].valid := 1, [287].log_data[2].valid := 1, [287].log_data[3].valid := 1, [287].log_data[4].valid := 1, [287].log_data[5].valid := 1, [287].log_data[6].valid := 1, [287].log_data[7].valid := 1, [287].log_data[8].valid := 1, [287].log_data[9].valid := 1, [287].log_data[10].valid := 1, [287].log_data[11].valid := 1, [287].log_data[12].valid := 1, [287].log_data[13].valid := 1, [287].log_data[14].valid := 1, [287].log_data[15].valid := 1, [287].log_data[16].valid := 1, [287].log_data[17].valid := 1, [287].log_data[18].valid := 1, [287].log_data[19].valid := 1, [287].time.Year := 2023, [287].time.Month := 1, [287].time.Day := 19, [287].time.Minute := 14, [287].time.Second := 59,
        [288].log_data[0].min := 1.0, [288].log_data[0].max := 1.0, [288].log_data[0].total := 900.0, [288].log_data[0].time := 900.0, [288].log_data[0].minminute := 15, [288].log_data[0].maxminute := 15, [288].log_data[0].valid := 1, [288].log_data[1].valid := 1, [288].log_data[2].valid := 1, [288].log_data[3].valid := 1, [288].log_data[4].valid := 1, [288].log_data[5].valid := 1, [288].log_data[6].valid := 1, [288].log_data[7].valid := 1, [288].log_data[8].valid := 1, [288].log_data[9].valid := 1, [288].log_data[10].valid := 1, [288].log_data[11].valid := 1, [288].log_data[12].valid := 1, [288].log_data[13].valid := 1, [288].log_data[14].valid := 1, [288].log_data[15].valid := 1, [288].log_data[16].valid := 1, [288].log_data[17].valid := 1, [288].log_data[18].valid := 1, [288].log_data[19].valid := 1, [288].time.Year := 2023, [288].time.Month := 1, [288].time.Day := 19, [288].time.Minute := 29, [288].time.Second := 59, [289].log_data[0].min := 1.0, [289].log_data[0].max := 1.0, [289].log_data[0].total := 900.0, [289].log_data[0].time := 900.0, [289].log_data[0].minminute := 30, [289].log_data[0].maxminute := 30, [289].log_data[0].valid := 1, [289].log_data[1].valid := 1, [289].log_data[2].valid := 1, [289].log_data[3].valid := 1, [289].log_data[4].valid := 1, [289].log_data[5].valid := 1, [289].log_data[6].valid := 1, [289].log_data[7].valid := 1, [289].log_data[8].valid := 1, [289].log_data[9].valid := 1, [289].log_data[10].valid := 1, [289].log_data[11].valid := 1, [289].log_data[12].valid := 1, [289].log_data[13].valid := 1, [289].log_data[14].valid := 1, [289].log_data[15].valid := 1, [289].log_data[16].valid := 1, [289].log_data[17].valid := 1, [289].log_data[18].valid := 1, [289].log_data[19].valid := 1, [289].time.Year := 2023, [289].time.Month := 1, [289].time.Day := 19,
        [289].time.Minute := 44, [289].time.Second := 59, [290].log_data[0].min := 1.0, [290].log_data[0].max := 1.0, [290].log_data[0].total := 900.0, [290].log_data[0].time := 900.0, [290].log_data[0].minminute := 45, [290].log_data[0].maxminute := 45, [290].log_data[0].valid := 1, [290].log_data[1].valid := 1, [290].log_data[2].valid := 1, [290].log_data[3].valid := 1, [290].log_data[4].valid := 1, [290].log_data[5].valid := 1, [290].log_data[6].valid := 1, [290].log_data[7].valid := 1, [290].log_data[8].valid := 1, [290].log_data[9].valid := 1, [290].log_data[10].valid := 1, [290].log_data[11].valid := 1, [290].log_data[12].valid := 1, [290].log_data[13].valid := 1, [290].log_data[14].valid := 1, [290].log_data[15].valid := 1, [290].log_data[16].valid := 1, [290].log_data[17].valid := 1, [290].log_data[18].valid := 1, [290].log_data[19].valid := 1, [290].time.Year := 2023, [290].time.Month := 1, [290].time.Day := 19, [290].time.Minute := 59, [290].time.Second := 59, [291].log_data[0].min := 1.0, [291].log_data[0].max := 1.0, [291].log_data[0].total := 900.0, [291].log_data[0].time := 900.0, [291].log_data[0].valid := 1, [291].log_data[1].valid := 1, [291].log_data[2].valid := 1, [291].log_data[3].valid := 1, [291].log_data[4].valid := 1, [291].log_data[5].valid := 1, [291].log_data[6].valid := 1, [291].log_data[7].valid := 1, [291].log_data[8].valid := 1, [291].log_data[9].valid := 1, [291].log_data[10].valid := 1, [291].log_data[11].valid := 1, [291].log_data[12].valid := 1, [291].log_data[13].valid := 1, [291].log_data[14].valid := 1, [291].log_data[15].valid := 1, [291].log_data[16].valid := 1, [291].log_data[17].valid := 1, [291].log_data[18].valid := 1, [291].log_data[19].valid := 1, [291].time.Year := 2023, [291].time.Month := 1, [291].time.Day := 19,
        [291].time.Hour := 1, [291].time.Minute := 14, [291].time.Second := 59, [292].log_data[0].min := 1.0, [292].log_data[0].max := 1.0, [292].log_data[0].total := 900.0, [292].log_data[0].time := 900.0, [292].log_data[0].minminute := 15, [292].log_data[0].maxminute := 15, [292].log_data[0].valid := 1, [292].log_data[1].valid := 1, [292].log_data[2].valid := 1, [292].log_data[3].valid := 1, [292].log_data[4].valid := 1, [292].log_data[5].valid := 1, [292].log_data[6].valid := 1, [292].log_data[7].valid := 1, [292].log_data[8].valid := 1, [292].log_data[9].valid := 1, [292].log_data[10].valid := 1, [292].log_data[11].valid := 1, [292].log_data[12].valid := 1, [292].log_data[13].valid := 1, [292].log_data[14].valid := 1, [292].log_data[15].valid := 1, [292].log_data[16].valid := 1, [292].log_data[17].valid := 1, [292].log_data[18].valid := 1, [292].log_data[19].valid := 1, [292].time.Year := 2023, [292].time.Month := 1, [292].time.Day := 19, [292].time.Hour := 1, [292].time.Minute := 29, [292].time.Second := 59, [293].log_data[0].min := 1.0, [293].log_data[0].max := 1.0, [293].log_data[0].total := 900.0, [293].log_data[0].time := 900.0, [293].log_data[0].minminute := 30, [293].log_data[0].maxminute := 30, [293].log_data[0].valid := 1, [293].log_data[1].valid := 1, [293].log_data[2].valid := 1, [293].log_data[3].valid := 1, [293].log_data[4].valid := 1, [293].log_data[5].valid := 1, [293].log_data[6].valid := 1, [293].log_data[7].valid := 1, [293].log_data[8].valid := 1, [293].log_data[9].valid := 1, [293].log_data[10].valid := 1, [293].log_data[11].valid := 1, [293].log_data[12].valid := 1, [293].log_data[13].valid := 1, [293].log_data[14].valid := 1, [293].log_data[15].valid := 1, [293].log_data[16].valid := 1, [293].log_data[17].valid := 1, [293].log_data[18].valid := 1,
        [293].log_data[19].valid := 1, [293].time.Year := 2023, [293].time.Month := 1, [293].time.Day := 19, [293].time.Hour := 1, [293].time.Minute := 44, [293].time.Second := 59, [294].log_data[0].min := 1.0, [294].log_data[0].max := 1.0, [294].log_data[0].total := 900.0, [294].log_data[0].time := 900.0, [294].log_data[0].minminute := 45, [294].log_data[0].maxminute := 45, [294].log_data[0].valid := 1, [294].log_data[1].valid := 1, [294].log_data[2].valid := 1, [294].log_data[3].valid := 1, [294].log_data[4].valid := 1, [294].log_data[5].valid := 1, [294].log_data[6].valid := 1, [294].log_data[7].valid := 1, [294].log_data[8].valid := 1, [294].log_data[9].valid := 1, [294].log_data[10].valid := 1, [294].log_data[11].valid := 1, [294].log_data[12].valid := 1, [294].log_data[13].valid := 1, [294].log_data[14].valid := 1, [294].log_data[15].valid := 1, [294].log_data[16].valid := 1, [294].log_data[17].valid := 1, [294].log_data[18].valid := 1, [294].log_data[19].valid := 1, [294].time.Year := 2023, [294].time.Month := 1, [294].time.Day := 19, [294].time.Hour := 1, [294].time.Minute := 59, [294].time.Second := 59, [295].log_data[0].min := 1.0, [295].log_data[0].max := 1.0, [295].log_data[0].total := 900.0, [295].log_data[0].time := 900.0, [295].log_data[0].valid := 1, [295].log_data[1].valid := 1, [295].log_data[2].valid := 1, [295].log_data[3].valid := 1, [295].log_data[4].valid := 1, [295].log_data[5].valid := 1, [295].log_data[6].valid := 1, [295].log_data[7].valid := 1, [295].log_data[8].valid := 1, [295].log_data[9].valid := 1, [295].log_data[10].valid := 1, [295].log_data[11].valid := 1, [295].log_data[12].valid := 1, [295].log_data[13].valid := 1, [295].log_data[14].valid := 1, [295].log_data[15].valid := 1, [295].log_data[16].valid := 1,
        [295].log_data[17].valid := 1, [295].log_data[18].valid := 1, [295].log_data[19].valid := 1, [295].time.Year := 2023, [295].time.Month := 1, [295].time.Day := 19, [295].time.Hour := 2, [295].time.Minute := 14, [295].time.Second := 59, [296].log_data[0].min := 1.0, [296].log_data[0].max := 1.0, [296].log_data[0].total := 900.0, [296].log_data[0].time := 900.0, [296].log_data[0].minminute := 15, [296].log_data[0].maxminute := 15, [296].log_data[0].valid := 1, [296].log_data[1].valid := 1, [296].log_data[2].valid := 1, [296].log_data[3].valid := 1, [296].log_data[4].valid := 1, [296].log_data[5].valid := 1, [296].log_data[6].valid := 1, [296].log_data[7].valid := 1, [296].log_data[8].valid := 1, [296].log_data[9].valid := 1, [296].log_data[10].valid := 1, [296].log_data[11].valid := 1, [296].log_data[12].valid := 1, [296].log_data[13].valid := 1, [296].log_data[14].valid := 1, [296].log_data[15].valid := 1, [296].log_data[16].valid := 1, [296].log_data[17].valid := 1, [296].log_data[18].valid := 1, [296].log_data[19].valid := 1, [296].time.Year := 2023, [296].time.Month := 1, [296].time.Day := 19, [296].time.Hour := 2, [296].time.Minute := 29, [296].time.Second := 59, [297].log_data[0].min := 1.0, [297].log_data[0].max := 1.0, [297].log_data[0].total := 900.0, [297].log_data[0].time := 900.0, [297].log_data[0].minminute := 30, [297].log_data[0].maxminute := 30, [297].log_data[0].valid := 1, [297].log_data[1].valid := 1, [297].log_data[2].valid := 1, [297].log_data[3].valid := 1, [297].log_data[4].valid := 1, [297].log_data[5].valid := 1, [297].log_data[6].valid := 1, [297].log_data[7].valid := 1, [297].log_data[8].valid := 1, [297].log_data[9].valid := 1, [297].log_data[10].valid := 1, [297].log_data[11].valid := 1, [297].log_data[12].valid := 1,
        [297].log_data[13].valid := 1, [297].log_data[14].valid := 1, [297].log_data[15].valid := 1, [297].log_data[16].valid := 1, [297].log_data[17].valid := 1, [297].log_data[18].valid := 1, [297].log_data[19].valid := 1, [297].time.Year := 2023, [297].time.Month := 1, [297].time.Day := 19, [297].time.Hour := 2, [297].time.Minute := 44, [297].time.Second := 59, [298].log_data[0].min := 1.0, [298].log_data[0].max := 1.0, [298].log_data[0].total := 900.0, [298].log_data[0].time := 900.0, [298].log_data[0].minminute := 45, [298].log_data[0].maxminute := 45, [298].log_data[0].valid := 1, [298].log_data[1].valid := 1, [298].log_data[2].valid := 1, [298].log_data[3].valid := 1, [298].log_data[4].valid := 1, [298].log_data[5].valid := 1, [298].log_data[6].valid := 1, [298].log_data[7].valid := 1, [298].log_data[8].valid := 1, [298].log_data[9].valid := 1, [298].log_data[10].valid := 1, [298].log_data[11].valid := 1, [298].log_data[12].valid := 1, [298].log_data[13].valid := 1, [298].log_data[14].valid := 1, [298].log_data[15].valid := 1, [298].log_data[16].valid := 1, [298].log_data[17].valid := 1, [298].log_data[18].valid := 1, [298].log_data[19].valid := 1, [298].time.Year := 2023, [298].time.Month := 1, [298].time.Day := 19, [298].time.Hour := 2, [298].time.Minute := 59, [298].time.Second := 59, [299].log_data[0].min := 1.0, [299].log_data[0].max := 1.0, [299].log_data[0].total := 900.0, [299].log_data[0].time := 900.0, [299].log_data[0].valid := 1, [299].log_data[1].valid := 1, [299].log_data[2].valid := 1, [299].log_data[3].valid := 1, [299].log_data[4].valid := 1, [299].log_data[5].valid := 1, [299].log_data[6].valid := 1, [299].log_data[7].valid := 1, [299].log_data[8].valid := 1, [299].log_data[9].valid := 1, [299].log_data[10].valid := 1,
        [299].log_data[11].valid := 1, [299].log_data[12].valid := 1, [299].log_data[13].valid := 1, [299].log_data[14].valid := 1, [299].log_data[15].valid := 1, [299].log_data[16].valid := 1, [299].log_data[17].valid := 1, [299].log_data[18].valid := 1, [299].log_data[19].valid := 1, [299].time.Year := 2023, [299].time.Month := 1, [299].time.Day := 19, [299].time.Hour := 3, [299].time.Minute := 14, [299].time.Second := 59, [300].log_data[0].min := 1.0, [300].log_data[0].max := 1.0, [300].log_data[0].total := 900.0, [300].log_data[0].time := 900.0, [300].log_data[0].minminute := 15, [300].log_data[0].maxminute := 15, [300].log_data[0].valid := 1, [300].log_data[1].valid := 1, [300].log_data[2].valid := 1, [300].log_data[3].valid := 1, [300].log_data[4].valid := 1, [300].log_data[5].valid := 1, [300].log_data[6].valid := 1, [300].log_data[7].valid := 1, [300].log_data[8].valid := 1, [300].log_data[9].valid := 1, [300].log_data[10].valid := 1, [300].log_data[11].valid := 1, [300].log_data[12].valid := 1, [300].log_data[13].valid := 1, [300].log_data[14].valid := 1, [300].log_data[15].valid := 1, [300].log_data[16].valid := 1, [300].log_data[17].valid := 1, [300].log_data[18].valid := 1, [300].log_data[19].valid := 1, [300].time.Year := 2023, [300].time.Month := 1, [300].time.Day := 19, [300].time.Hour := 3, [300].time.Minute := 29, [300].time.Second := 59, [301].log_data[0].min := 1.0, [301].log_data[0].max := 1.0, [301].log_data[0].total := 900.0, [301].log_data[0].time := 900.0, [301].log_data[0].minminute := 30, [301].log_data[0].maxminute := 30, [301].log_data[0].valid := 1, [301].log_data[1].valid := 1, [301].log_data[2].valid := 1, [301].log_data[3].valid := 1, [301].log_data[4].valid := 1, [301].log_data[5].valid := 1, [301].log_data[6].valid := 1,
        [301].log_data[7].valid := 1, [301].log_data[8].valid := 1, [301].log_data[9].valid := 1, [301].log_data[10].valid := 1, [301].log_data[11].valid := 1, [301].log_data[12].valid := 1, [301].log_data[13].valid := 1, [301].log_data[14].valid := 1, [301].log_data[15].valid := 1, [301].log_data[16].valid := 1, [301].log_data[17].valid := 1, [301].log_data[18].valid := 1, [301].log_data[19].valid := 1, [301].time.Year := 2023, [301].time.Month := 1, [301].time.Day := 19, [301].time.Hour := 3, [301].time.Minute := 44, [301].time.Second := 59, [302].log_data[0].min := 1.0, [302].log_data[0].max := 1.0, [302].log_data[0].total := 900.0, [302].log_data[0].time := 900.0, [302].log_data[0].minminute := 45, [302].log_data[0].maxminute := 45, [302].log_data[0].valid := 1, [302].log_data[1].valid := 1, [302].log_data[2].valid := 1, [302].log_data[3].valid := 1, [302].log_data[4].valid := 1, [302].log_data[5].valid := 1, [302].log_data[6].valid := 1, [302].log_data[7].valid := 1, [302].log_data[8].valid := 1, [302].log_data[9].valid := 1, [302].log_data[10].valid := 1, [302].log_data[11].valid := 1, [302].log_data[12].valid := 1, [302].log_data[13].valid := 1, [302].log_data[14].valid := 1, [302].log_data[15].valid := 1, [302].log_data[16].valid := 1, [302].log_data[17].valid := 1, [302].log_data[18].valid := 1, [302].log_data[19].valid := 1, [302].time.Year := 2023, [302].time.Month := 1, [302].time.Day := 19, [302].time.Hour := 3, [302].time.Minute := 59, [302].time.Second := 59, [303].log_data[0].min := 1.0, [303].log_data[0].max := 1.0, [303].log_data[0].total := 900.0, [303].log_data[0].time := 900.0, [303].log_data[0].valid := 1, [303].log_data[1].valid := 1, [303].log_data[2].valid := 1, [303].log_data[3].valid := 1, [303].log_data[4].valid := 1,
        [303].log_data[5].valid := 1, [303].log_data[6].valid := 1, [303].log_data[7].valid := 1, [303].log_data[8].valid := 1, [303].log_data[9].valid := 1, [303].log_data[10].valid := 1, [303].log_data[11].valid := 1, [303].log_data[12].valid := 1, [303].log_data[13].valid := 1, [303].log_data[14].valid := 1, [303].log_data[15].valid := 1, [303].log_data[16].valid := 1, [303].log_data[17].valid := 1, [303].log_data[18].valid := 1, [303].log_data[19].valid := 1, [303].time.Year := 2023, [303].time.Month := 1, [303].time.Day := 19, [303].time.Hour := 4, [303].time.Minute := 14, [303].time.Second := 59, [304].log_data[0].min := 1.0, [304].log_data[0].max := 1.0, [304].log_data[0].total := 900.0, [304].log_data[0].time := 900.0, [304].log_data[0].minminute := 15, [304].log_data[0].maxminute := 15, [304].log_data[0].valid := 1, [304].log_data[1].valid := 1, [304].log_data[2].valid := 1, [304].log_data[3].valid := 1, [304].log_data[4].valid := 1, [304].log_data[5].valid := 1, [304].log_data[6].valid := 1, [304].log_data[7].valid := 1, [304].log_data[8].valid := 1, [304].log_data[9].valid := 1, [304].log_data[10].valid := 1, [304].log_data[11].valid := 1, [304].log_data[12].valid := 1, [304].log_data[13].valid := 1, [304].log_data[14].valid := 1, [304].log_data[15].valid := 1, [304].log_data[16].valid := 1, [304].log_data[17].valid := 1, [304].log_data[18].valid := 1, [304].log_data[19].valid := 1, [304].time.Year := 2023, [304].time.Month := 1, [304].time.Day := 19, [304].time.Hour := 4, [304].time.Minute := 29, [304].time.Second := 59, [305].log_data[0].min := 1.0, [305].log_data[0].max := 1.0, [305].log_data[0].total := 900.0, [305].log_data[0].time := 900.0, [305].log_data[0].minminute := 30, [305].log_data[0].maxminute := 30, [305].log_data[0].valid := 1,
        [305].log_data[1].valid := 1, [305].log_data[2].valid := 1, [305].log_data[3].valid := 1, [305].log_data[4].valid := 1, [305].log_data[5].valid := 1, [305].log_data[6].valid := 1, [305].log_data[7].valid := 1, [305].log_data[8].valid := 1, [305].log_data[9].valid := 1, [305].log_data[10].valid := 1, [305].log_data[11].valid := 1, [305].log_data[12].valid := 1, [305].log_data[13].valid := 1, [305].log_data[14].valid := 1, [305].log_data[15].valid := 1, [305].log_data[16].valid := 1, [305].log_data[17].valid := 1, [305].log_data[18].valid := 1, [305].log_data[19].valid := 1, [305].time.Year := 2023, [305].time.Month := 1, [305].time.Day := 19, [305].time.Hour := 4, [305].time.Minute := 44, [305].time.Second := 59, [306].log_data[0].min := 1.0, [306].log_data[0].max := 1.0, [306].log_data[0].total := 900.0, [306].log_data[0].time := 900.0, [306].log_data[0].minminute := 45, [306].log_data[0].maxminute := 45, [306].log_data[0].valid := 1, [306].log_data[1].valid := 1, [306].log_data[2].valid := 1, [306].log_data[3].valid := 1, [306].log_data[4].valid := 1, [306].log_data[5].valid := 1, [306].log_data[6].valid := 1, [306].log_data[7].valid := 1, [306].log_data[8].valid := 1, [306].log_data[9].valid := 1, [306].log_data[10].valid := 1, [306].log_data[11].valid := 1, [306].log_data[12].valid := 1, [306].log_data[13].valid := 1, [306].log_data[14].valid := 1, [306].log_data[15].valid := 1, [306].log_data[16].valid := 1, [306].log_data[17].valid := 1, [306].log_data[18].valid := 1, [306].log_data[19].valid := 1, [306].time.Year := 2023, [306].time.Month := 1, [306].time.Day := 19, [306].time.Hour := 4, [306].time.Minute := 59, [306].time.Second := 59, [307].log_data[0].min := 1.0, [307].log_data[0].max := 1.0, [307].log_data[0].total := 900.0,
